C03649=1150.489,20.395,-48.948,179.944,6.210,149.138
C03650=1150.495,20.146,-48.934,179.942,6.210,149.139
C03651=1150.499,19.897,-48.920,179.939,6.209,149.139
C03652=1150.504,19.647,-48.905,179.936,6.208,149.140
C03653=1150.509,19.397,-48.891,179.934,6.207,149.141
C03654=1150.514,19.147,-48.877,179.931,6.206,149.141
C03655=1150.520,18.898,-48.863,179.929,6.205,149.142
C03656=1150.525,18.649,-48.849,179.926,6.204,149.142
C03657=1150.530,18.399,-48.834,179.924,6.203,149.143
C03658=1150.535,18.150,-48.820,179.922,6.203,149.143
C03659=1150.541,17.900,-48.807,179.919,6.202,149.144
C03660=1150.546,17.650,-48.793,179.916,6.200,149.145
C03661=1150.551,17.400,-48.778,179.914,6.200,149.145
C03662=1150.556,17.151,-48.764,179.911,6.199,149.146
C03663=1150.561,16.902,-48.750,179.909,6.199,149.146
C03664=1150.566,16.652,-48.736,179.906,6.197,149.147
C03665=1150.571,16.402,-48.722,179.903,6.197,149.147
C03666=1150.576,16.153,-48.708,179.901,6.196,149.148
C03667=1150.581,15.904,-48.694,179.898,6.195,149.149
C03668=1150.586,15.653,-48.680,179.896,6.194,149.149
C03669=1150.592,15.404,-48.667,179.894,6.193,149.150
C03670=1150.596,15.155,-48.652,179.891,6.193,149.150
C03671=1150.601,14.905,-48.638,179.889,6.192,149.151
C03672=1150.607,14.656,-48.624,179.885,6.190,149.151
C03673=1150.612,14.406,-48.611,179.883,6.190,149.152
C03674=1150.616,14.156,-48.597,179.881,6.189,149.152
C03675=1150.622,13.907,-48.583,179.878,6.188,149.153
C03676=1150.627,13.657,-48.569,179.875,6.187,149.154
C03677=1150.632,13.408,-48.554,179.873,6.186,149.154
C03678=1150.638,13.158,-48.541,179.870,6.186,149.155
C03679=1150.642,12.909,-48.527,179.868,6.185,149.155
C03680=1150.647,12.659,-48.513,179.866,6.185,149.156
C03681=1150.653,12.410,-48.499,179.863,6.183,149.156
C03682=1150.658,12.160,-48.486,179.861,6.182,149.157
C03683=1150.663,11.910,-48.471,179.858,6.182,149.158
C03684=1150.668,11.661,-48.458,179.856,6.181,149.158
C03685=1150.673,11.411,-48.445,179.853,6.180,149.159
C03686=1150.678,11.162,-48.431,179.850,6.179,149.159
C03687=1150.683,10.912,-48.416,179.848,6.178,149.160
C03688=1150.688,10.662,-48.403,179.846,6.177,149.160
C03689=1150.693,10.413,-48.390,179.843,6.177,149.161
C03690=1150.698,10.164,-48.375,179.840,6.175,149.161
C03691=1150.704,9.913,-48.362,179.838,6.175,149.162
C03692=1150.708,9.664,-48.348,179.835,6.174,149.163
C03693=1150.713,9.415,-48.334,179.833,6.174,149.163
C03694=1150.719,9.165,-48.321,179.831,6.173,149.164
C03695=1150.724,8.915,-48.307,179.827,6.172,149.164
C03696=1150.729,8.666,-48.294,179.825,6.171,149.165
C03697=1150.734,8.416,-48.280,179.823,6.170,149.165
C03698=1150.739,8.167,-48.265,179.820,6.170,149.166
C03699=1150.744,7.917,-48.253,179.818,6.169,149.166
C03700=1150.749,7.668,-48.239,179.815,6.167,149.167
C03701=1150.755,7.418,-48.225,179.813,6.167,149.168
C03702=1150.759,7.169,-48.212,179.810,6.166,149.168
C03703=1150.765,6.919,-48.198,179.808,6.165,149.169
C03704=1150.770,6.669,-48.184,179.805,6.165,149.169
C03705=1150.775,6.419,-48.171,179.802,6.163,149.170
C03706=1150.780,6.170,-48.157,179.800,6.163,149.171
C03707=1150.786,5.920,-48.144,179.798,6.162,149.171
C03708=1150.790,5.671,-48.130,179.795,6.162,149.172
C03709=1150.796,5.421,-48.117,179.793,6.161,149.172
C03710=1150.800,5.172,-48.104,179.790,6.160,149.173
C03711=1150.806,4.922,-48.090,179.787,6.159,149.173
C03712=1150.811,4.673,-48.076,179.785,6.158,149.174
C03713=1150.816,4.423,-48.063,179.783,6.158,149.175
C03714=1150.821,4.174,-48.049,179.780,6.157,149.175
C03715=1150.826,3.924,-48.036,179.778,6.156,149.176
C03716=1150.831,3.675,-48.022,179.776,6.155,149.176
C03717=1150.837,3.424,-48.009,179.772,6.154,149.177
C03718=1150.842,3.175,-47.996,179.770,6.153,149.177
C03719=1150.847,2.925,-47.982,179.767,6.153,149.178
C03720=1150.852,2.676,-47.969,179.765,6.152,149.178
C03721=1150.857,2.426,-47.955,179.763,6.152,149.179
C03722=1150.862,2.177,-47.942,179.760,6.151,149.180
C03723=1150.867,1.908,-47.927,179.757,6.150,149.180
C03724=1150.873,1.638,-47.913,179.755,6.149,149.181
C03725=1150.879,1.369,-47.899,179.752,6.148,149.181
C03726=1150.884,1.099,-47.885,179.749,6.147,149.182
C03727=1150.889,0.850,-47.871,179.747,6.146,149.183
C03728=1150.894,0.600,-47.858,179.744,6.146,149.183
C03729=1150.900,0.351,-47.845,179.742,6.145,149.184
C03730=1150.905,0.101,-47.832,179.739,6.145,149.184
C03731=1150.910,-0.148,-47.818,179.737,6.144,149.185
C03732=1150.915,-0.398,-47.805,179.734,6.143,149.186
C03733=1150.921,-0.648,-47.792,179.732,6.142,149.186
C03734=1150.925,-0.898,-47.778,179.729,6.141,149.187
C03735=1150.931,-1.147,-47.765,179.727,6.141,149.187
C03736=1150.936,-1.396,-47.752,179.724,6.140,149.188
C03737=1150.941,-1.647,-47.739,179.722,6.139,149.188
C03738=1150.946,-1.895,-47.725,179.720,6.139,149.189
C03739=1150.951,-2.146,-47.712,179.717,6.137,149.189
C03740=1150.956,-2.395,-47.699,179.715,6.136,149.190
C03741=1150.961,-2.644,-47.687,179.712,6.136,149.191
C03742=1150.967,-2.895,-47.673,179.710,6.135,149.191
C03743=1150.971,-3.143,-47.660,179.707,6.135,149.192
C03744=1150.977,-3.394,-47.646,179.705,6.134,149.192
C03745=1150.982,-3.643,-47.634,179.702,6.133,149.193
C03746=1150.988,-3.893,-47.620,179.700,6.133,149.193
C03747=1150.992,-4.143,-47.607,179.697,6.131,149.194
C03748=1150.997,-4.392,-47.595,179.695,6.131,149.195
C03749=1151.003,-4.641,-47.581,179.692,6.130,149.195
C03750=1151.007,-4.891,-47.568,179.690,6.129,149.196
C03751=1151.013,-5.140,-47.555,179.687,6.129,149.196
C03752=1151.018,-5.391,-47.542,179.685,6.128,149.197
C03753=1151.023,-5.640,-47.529,179.682,6.128,149.198
C03754=1151.029,-5.890,-47.516,179.680,6.127,149.198
C03755=1151.033,-6.140,-47.503,179.677,6.126,149.199
C03756=1151.038,-6.389,-47.490,179.675,6.125,149.199
C03757=1151.044,-6.639,-47.477,179.672,6.124,149.200
C03758=1151.049,-6.888,-47.464,179.670,6.124,149.200
C03759=1151.054,-7.137,-47.451,179.668,6.123,149.201
C03760=1151.060,-7.387,-47.438,179.665,6.122,149.202
C03761=1151.064,-7.637,-47.425,179.663,6.122,149.202
C03762=1151.069,-7.886,-47.412,179.660,6.121,149.203
C03763=1151.074,-8.136,-47.400,179.658,6.120,149.203
C03764=1151.080,-8.386,-47.386,179.655,6.120,149.204
C03765=1151.085,-8.635,-47.373,179.653,6.119,149.204
C03766=1151.090,-8.885,-47.361,179.650,6.118,149.205
C03767=1151.096,-9.134,-47.348,179.648,6.117,149.205
C03768=1151.100,-9.384,-47.335,179.645,6.117,149.206
C03769=1151.105,-9.634,-47.322,179.643,6.116,149.207
C03770=1151.110,-9.883,-47.309,179.640,6.115,149.207
C03771=1151.116,-10.133,-47.296,179.638,6.115,149.208
C03772=1151.121,-10.383,-47.283,179.635,6.114,149.208
C03773=1151.126,-10.632,-47.271,179.633,6.113,149.209
C03774=1151.131,-10.882,-47.259,179.631,6.113,149.210
C03775=1151.136,-11.132,-47.246,179.628,6.112,149.210
C03776=1151.142,-11.381,-47.233,179.626,6.111,149.211
C03777=1151.147,-11.631,-47.220,179.624,6.111,149.211
C03778=1151.152,-11.880,-47.207,179.621,6.110,149.212
C03779=1151.157,-12.130,-47.194,179.618,6.109,149.212
C03780=1151.162,-12.380,-47.181,179.616,6.108,149.213
C03781=1151.167,-12.629,-47.169,179.613,6.108,149.214
C03782=1151.173,-12.878,-47.156,179.611,6.107,149.214
C03783=1151.177,-13.128,-47.143,179.608,6.106,149.215
C03784=1151.183,-13.378,-47.131,179.606,6.105,149.215
C03785=1151.188,-13.628,-47.119,179.604,6.105,149.216
C03786=1151.194,-13.877,-47.105,179.601,6.104,149.216
C03787=1151.198,-14.127,-47.092,179.599,6.104,149.217
C03788=1151.203,-14.377,-47.080,179.597,6.103,149.218
C03789=1151.209,-14.627,-47.068,179.594,6.103,149.218
C03790=1151.214,-14.876,-47.055,179.592,6.102,149.219
C03791=1151.219,-15.125,-47.043,179.589,6.101,149.219
C03792=1151.223,-15.375,-47.030,179.587,6.101,149.220
C03793=1151.229,-15.625,-47.017,179.584,6.100,149.221
C03794=1151.235,-15.875,-47.005,179.582,6.099,149.221
C03795=1151.240,-16.124,-46.992,179.580,6.098,149.221
C03796=1151.245,-16.373,-46.980,179.577,6.097,149.222
C03797=1151.250,-16.623,-46.967,179.575,6.096,149.223
C03798=1151.255,-16.873,-46.955,179.572,6.096,149.223
C03799=1151.260,-17.123,-46.942,179.570,6.095,149.224
C03800=1151.265,-17.372,-46.929,179.567,6.095,149.225
C03801=1151.270,-17.621,-46.917,179.565,6.094,149.225
C03802=1151.276,-17.871,-46.905,179.562,6.094,149.226
C03803=1151.282,-18.121,-46.892,179.560,6.093,149.226
C03804=1151.286,-18.371,-46.879,179.557,6.092,149.227
C03805=1151.292,-18.621,-46.867,179.555,6.092,149.227
C03806=1151.297,-18.870,-46.854,179.552,6.091,149.228
C03807=1151.302,-19.119,-46.842,179.550,6.090,149.228
C03808=1151.307,-19.369,-46.830,179.548,6.090,149.229
C03809=1151.312,-19.619,-46.817,179.545,6.089,149.230
C03810=1151.317,-19.868,-46.805,179.543,6.088,149.230
C03811=1151.322,-20.119,-46.792,179.541,6.088,149.231
C03812=1151.327,-20.368,-46.780,179.538,6.087,149.231
C03813=1151.333,-20.618,-46.768,179.536,6.087,149.232
C03814=1151.338,-20.867,-46.755,179.534,6.086,149.232
C03815=1151.343,-21.117,-46.743,179.531,6.085,149.233
C03816=1151.348,-21.367,-46.731,179.529,6.085,149.234
C03817=1151.354,-21.616,-46.718,179.526,6.084,149.234
C03818=1151.359,-21.866,-46.706,179.524,6.083,149.235
C03819=1151.364,-22.115,-46.694,179.521,6.083,149.235
C03820=1151.369,-22.364,-46.681,179.519,6.082,149.236
C03821=1151.375,-22.614,-46.669,179.516,6.082,149.237
C03822=1151.379,-22.864,-46.656,179.514,6.081,149.237
C03823=1151.385,-23.114,-46.644,179.512,6.081,149.238
C03824=1151.390,-23.364,-46.632,179.509,6.080,149.238
C03825=1151.395,-23.614,-46.620,179.507,6.079,149.239
C03826=1151.400,-23.863,-46.607,179.505,6.079,149.239
C03827=1151.406,-24.133,-46.595,179.502,6.078,149.240
C03828=1151.412,-24.403,-46.582,179.499,6.076,149.241
C03829=1151.417,-24.673,-46.568,179.496,6.076,149.241
C03830=1151.423,-24.943,-46.555,179.494,6.076,149.242
C03831=1151.428,-25.192,-46.544,179.492,6.075,149.242
C03832=1151.433,-25.442,-46.531,179.489,6.074,149.243
C03833=1151.438,-25.691,-46.519,179.487,6.074,149.244
C03834=1151.443,-25.941,-46.506,179.485,6.073,149.244
C03835=1151.448,-26.191,-46.494,179.482,6.072,149.245
C03836=1151.454,-26.441,-46.482,179.480,6.072,149.245
C03837=1151.459,-26.691,-46.470,179.477,6.071,149.246
C03838=1151.464,-26.941,-46.458,179.475,6.070,149.246
C03839=1151.469,-27.190,-46.446,179.472,6.070,149.247
C03840=1151.474,-27.440,-46.434,179.470,6.069,149.248
C03841=1151.479,-27.689,-46.421,179.467,6.069,149.248
C03842=1151.485,-27.939,-46.409,179.465,6.068,149.249
C03843=1151.490,-28.189,-46.398,179.463,6.068,149.249
C03844=1151.495,-28.438,-46.385,179.460,6.067,149.250
C03845=1151.500,-28.688,-46.374,179.458,6.066,149.251
C03846=1151.505,-28.938,-46.362,179.455,6.066,149.251
C03847=1151.511,-29.187,-46.349,179.453,6.065,149.252
C03848=1151.516,-29.437,-46.337,179.451,6.064,149.252
C03849=1151.521,-29.687,-46.325,179.449,6.064,149.253
C03850=1151.526,-29.936,-46.313,179.446,6.064,149.253
C03851=1151.531,-30.186,-46.302,179.444,6.063,149.254
C03852=1151.537,-30.436,-46.290,179.442,6.063,149.255
C03853=1151.542,-30.684,-46.277,179.439,6.062,149.255
C03854=1151.548,-30.934,-46.266,179.437,6.061,149.256
C03855=1151.553,-31.184,-46.254,179.435,6.061,149.256
C03856=1151.558,-31.434,-46.242,179.432,6.060,149.257
C03857=1151.563,-31.683,-46.230,179.430,6.059,149.257
C03858=1151.569,-31.933,-46.218,179.427,6.059,149.258
C03859=1151.573,-32.183,-46.207,179.425,6.058,149.259
C03860=1151.579,-32.433,-46.195,179.423,6.057,149.259
C03861=1151.584,-32.682,-46.182,179.420,6.057,149.260
C03862=1151.589,-32.932,-46.170,179.418,6.056,149.260
C03863=1151.594,-33.181,-46.159,179.415,6.056,149.261
C03864=1151.599,-33.431,-46.147,179.413,6.055,149.261
C03865=1151.604,-33.681,-46.134,179.410,6.055,149.262
C03866=1151.609,-33.930,-46.123,179.408,6.054,149.263
C03867=1151.615,-34.180,-46.111,179.405,6.053,149.263
C03868=1151.621,-34.430,-46.100,179.403,6.053,149.264
C03869=1151.625,-34.679,-46.088,179.401,6.052,149.264
C03870=1151.631,-34.929,-46.077,179.398,6.051,149.265
C03871=1151.636,-35.178,-46.064,179.397,6.051,149.265
C03872=1151.641,-35.428,-46.052,179.394,6.051,149.266
C03873=1151.646,-35.678,-46.041,179.392,6.050,149.267
C03874=1151.651,-35.928,-46.029,179.389,6.050,149.267
C03875=1151.657,-36.178,-46.017,179.387,6.049,149.268
C03876=1151.662,-36.427,-46.006,179.384,6.049,149.268
C03877=1151.668,-36.677,-45.994,179.382,6.048,149.269
C03878=1151.672,-36.926,-45.983,179.380,6.047,149.270
C03879=1151.678,-37.176,-45.971,179.377,6.047,149.270
C03880=1151.683,-37.426,-45.958,179.375,6.046,149.271
C03881=1151.687,-37.675,-45.947,179.373,6.045,149.271
C03882=1151.693,-37.925,-45.935,179.370,6.045,149.272
C03883=1151.699,-38.174,-45.924,179.368,6.044,149.272
C03884=1151.704,-38.424,-45.912,179.366,6.044,149.273
C03885=1151.709,-38.674,-45.901,179.363,6.044,149.274
C03886=1151.714,-38.924,-45.889,179.361,6.043,149.274
C03887=1151.719,-39.174,-45.877,179.359,6.043,149.275
C03888=1151.725,-39.423,-45.866,179.356,6.042,149.275
C03889=1151.730,-39.672,-45.855,179.354,6.041,149.276
C03890=1151.735,-39.922,-45.843,179.352,6.041,149.276
C03891=1151.740,-40.172,-45.831,179.349,6.040,149.277
C03892=1151.745,-40.422,-45.820,179.347,6.039,149.278
C03893=1151.751,-40.672,-45.808,179.345,6.039,149.278
C03894=1151.756,-40.921,-45.797,179.342,6.038,149.279
C03895=1151.762,-41.171,-45.785,179.340,6.037,149.279
C03896=1151.766,-41.420,-45.774,179.338,6.038,149.280
C03897=1151.772,-41.670,-45.762,179.335,6.037,149.280
C03898=1151.776,-41.920,-45.750,179.333,6.036,149.281
C03899=1151.782,-42.169,-45.739,179.331,6.036,149.282
C03900=1151.787,-42.419,-45.728,179.328,6.035,149.282
C03901=1151.793,-42.669,-45.716,179.326,6.035,149.283
C03902=1151.798,-42.919,-45.705,179.324,6.034,149.283
C03903=1151.803,-43.169,-45.693,179.321,6.033,149.284
C03904=1151.808,-43.418,-45.682,179.319,6.033,149.284
C03905=1151.814,-43.668,-45.670,179.317,6.033,149.285
C03906=1151.818,-43.917,-45.659,179.314,6.032,149.286
C03907=1151.824,-44.167,-45.647,179.312,6.031,149.286
C03908=1151.829,-44.416,-45.636,179.310,6.031,149.287
C03909=1151.835,-44.667,-45.625,179.307,6.030,149.287
C03910=1151.840,-44.916,-45.614,179.305,6.030,149.288
C03911=1151.845,-45.166,-45.602,179.303,6.029,149.288
C03912=1151.850,-45.415,-45.591,179.300,6.029,149.289
C03913=1151.855,-45.665,-45.580,179.298,6.028,149.290
C03914=1151.860,-45.915,-45.568,179.296,6.028,149.290
C03915=1151.865,-46.165,-45.557,179.293,6.027,149.291
C03916=1151.871,-46.414,-45.546,179.291,6.027,149.291
C03917=1151.876,-46.664,-45.535,179.289,6.026,149.292
C03918=1151.882,-46.914,-45.523,179.286,6.025,149.293
C03919=1151.887,-47.163,-45.512,179.284,6.025,149.293
C03920=1151.892,-47.413,-45.501,179.282,6.024,149.294
C03921=1151.897,-47.663,-45.489,179.279,6.024,149.294
C03922=1151.902,-47.913,-45.478,179.277,6.024,149.295
C03923=1151.908,-48.162,-45.466,179.275,6.023,149.295
C03924=1151.913,-48.412,-45.456,179.272,6.023,149.296
C03925=1151.918,-48.662,-45.445,179.270,6.022,149.297
C03926=1151.924,-48.911,-45.433,179.268,6.022,149.297
C03927=1151.928,-49.161,-45.422,179.265,6.021,149.298
C03928=1151.934,-49.411,-45.411,179.263,6.020,149.298
C03929=1151.939,-49.660,-45.400,179.261,6.020,149.299
C03930=1151.944,-49.910,-45.388,179.259,6.020,149.299
C03931=1151.950,-50.181,-45.376,179.256,6.019,149.300
C03932=1151.956,-50.451,-45.364,179.254,6.019,149.301
C03933=1151.962,-50.722,-45.352,179.251,6.018,149.301
C03934=1151.967,-50.993,-45.340,179.249,6.018,149.302
C03935=1151.972,-51.242,-45.329,179.247,6.017,149.302
C03936=1151.977,-51.492,-45.318,179.244,6.016,149.303
C03937=1151.983,-51.742,-45.306,179.242,6.016,149.304
C03938=1151.988,-51.991,-45.295,179.239,6.015,149.304
C03939=1151.993,-52.241,-45.285,179.237,6.014,149.305
C03940=1151.998,-52.490,-45.274,179.235,6.014,149.305
C03941=1152.004,-52.741,-45.263,179.233,6.014,149.306
C03942=1152.009,-52.990,-45.251,179.230,6.013,149.306
C03943=1152.014,-53.239,-45.241,179.228,6.013,149.307
C03944=1152.020,-53.490,-45.229,179.226,6.012,149.308
C03945=1152.025,-53.739,-45.218,179.223,6.012,149.308
C03946=1152.030,-53.989,-45.208,179.221,6.012,149.309
C03947=1152.035,-54.239,-45.197,179.219,6.011,149.309
C03948=1152.041,-54.488,-45.186,179.216,6.010,149.310
C03949=1152.046,-54.738,-45.174,179.214,6.010,149.310
C03950=1152.051,-54.988,-45.163,179.212,6.009,149.311
C03951=1152.056,-55.237,-45.153,179.209,6.009,149.312
C03952=1152.062,-55.487,-45.141,179.208,6.009,149.312
C03953=1152.067,-55.737,-45.131,179.205,6.008,149.313
C03954=1152.072,-55.986,-45.120,179.203,6.007,149.313
C03955=1152.077,-56.237,-45.109,179.200,6.007,149.314
C03956=1152.082,-56.485,-45.098,179.198,6.006,149.315
C03957=1152.088,-56.736,-45.087,179.195,6.006,149.315
C03958=1152.093,-56.985,-45.076,179.194,6.006,149.316
C03959=1152.098,-57.235,-45.065,179.192,6.005,149.316
C03960=1152.103,-57.485,-45.054,179.189,6.005,149.317
C03961=1152.109,-57.734,-45.044,179.187,6.004,149.317
C03962=1152.113,-57.984,-45.033,179.184,6.003,149.318
C03963=1152.120,-58.234,-45.022,179.183,6.003,149.319
C03964=1152.125,-58.484,-45.011,179.180,6.003,149.319
C03965=1152.130,-58.733,-45.000,179.178,6.002,149.320
C03966=1152.135,-58.983,-44.990,179.176,6.001,149.320
C03967=1152.140,-59.232,-44.979,179.173,6.001,149.321
C03968=1152.145,-59.482,-44.968,179.171,6.001,149.321
C03969=1152.151,-59.732,-44.956,179.169,6.000,149.322
C03970=1152.156,-59.982,-44.946,179.166,6.000,149.323
C03971=1152.161,-60.232,-44.936,179.164,5.999,149.323
C03972=1152.166,-60.481,-44.925,179.162,5.999,149.324
C03973=1152.171,-60.731,-44.914,179.160,5.999,149.324
C03974=1152.177,-60.981,-44.904,179.158,5.998,149.325
C03975=1152.182,-61.230,-44.893,179.155,5.998,149.325
C03976=1152.187,-61.480,-44.882,179.153,5.997,149.326
C03977=1152.192,-61.730,-44.871,179.150,5.996,149.327
C03978=1152.198,-61.979,-44.860,179.149,5.996,149.327
C03979=1152.203,-62.230,-44.850,179.146,5.996,149.328
C03980=1152.209,-62.479,-44.839,179.144,5.995,149.328
C03981=1152.214,-62.729,-44.828,179.142,5.994,149.329
C03982=1152.219,-62.978,-44.818,179.139,5.994,149.329
C03983=1152.224,-63.229,-44.807,179.137,5.994,149.330
C03984=1152.230,-63.478,-44.797,179.135,5.993,149.330
C03985=1152.235,-63.728,-44.786,179.132,5.993,149.331
C03986=1152.240,-63.977,-44.776,179.130,5.992,149.332
C03987=1152.245,-64.227,-44.764,179.128,5.992,149.332
C03988=1152.250,-64.477,-44.754,179.126,5.992,149.333
C03989=1152.256,-64.726,-44.744,179.124,5.991,149.333
C03990=1152.261,-64.976,-44.733,179.121,5.991,149.334
C03991=1152.266,-65.225,-44.723,179.119,5.990,149.334
C03992=1152.271,-65.476,-44.712,179.117,5.990,149.335
C03993=1152.277,-65.725,-44.702,179.115,5.989,149.336
C03994=1152.282,-65.975,-44.691,179.113,5.989,149.336
C03995=1152.288,-66.225,-44.681,179.110,5.988,149.337
C03996=1152.292,-66.474,-44.670,179.108,5.988,149.337
C03997=1152.298,-66.724,-44.659,179.106,5.988,149.338
C03998=1152.303,-66.974,-44.649,179.103,5.987,149.338
C03999=1152.308,-67.224,-44.639,179.101,5.986,149.339
C04000=1152.314,-67.473,-44.628,179.099,5.986,149.340
C04001=1152.319,-67.723,-44.617,179.097,5.986,149.340
C04002=1152.324,-67.973,-44.607,179.095,5.985,149.341
C04003=1152.329,-68.223,-44.596,179.092,5.985,149.341
C04004=1152.335,-68.472,-44.586,179.090,5.984,149.342
C04005=1152.341,-68.722,-44.576,179.088,5.984,149.342
C04006=1152.346,-68.972,-44.565,179.086,5.984,149.343
C04007=1152.351,-69.222,-44.555,179.083,5.983,149.343
C04008=1152.356,-69.471,-44.544,179.081,5.982,149.344
C04009=1152.361,-69.721,-44.534,179.079,5.983,149.345
C04010=1152.367,-69.970,-44.523,179.077,5.982,149.345
C04011=1152.372,-70.221,-44.513,179.074,5.981,149.346
C04012=1152.378,-70.470,-44.503,179.072,5.981,149.346
C04013=1152.383,-70.720,-44.493,179.071,5.981,149.347
C04014=1152.388,-70.970,-44.482,179.068,5.980,149.348
C04015=1152.394,-71.219,-44.472,179.066,5.979,149.348
C04016=1152.398,-71.469,-44.462,179.063,5.979,149.349
C04017=1152.404,-71.719,-44.452,179.061,5.979,149.349
C04018=1152.409,-71.968,-44.441,179.059,5.978,149.350
C04019=1152.414,-72.219,-44.431,179.057,5.978,149.350
C04020=1152.420,-72.468,-44.421,179.054,5.977,149.351
C04021=1152.425,-72.717,-44.410,179.053,5.977,149.351
C04022=1152.430,-72.967,-44.399,179.050,5.977,149.352
C04023=1152.436,-73.217,-44.389,179.048,5.976,149.353
C04024=1152.441,-73.466,-44.379,179.045,5.976,149.353
C04025=1152.446,-73.716,-44.369,179.044,5.976,149.354
C04026=1152.451,-73.966,-44.358,179.041,5.975,149.354
C04027=1152.457,-74.216,-44.348,179.039,5.974,149.355
C04028=1152.462,-74.466,-44.338,179.037,5.974,149.355
C04029=1152.468,-74.716,-44.328,179.035,5.974,149.356
C04030=1152.473,-74.965,-44.318,179.032,5.973,149.357
C04031=1152.478,-75.215,-44.308,179.030,5.973,149.357
C04032=1152.483,-75.465,-44.298,179.029,5.973,149.358
C04033=1152.489,-75.715,-44.288,179.026,5.972,149.358
C04034=1152.494,-75.964,-44.277,179.024,5.971,149.359
C04035=1152.500,-76.235,-44.266,179.021,5.971,149.359
C04036=1152.505,-76.507,-44.255,179.019,5.970,149.360
C04037=1152.511,-76.778,-44.244,179.017,5.971,149.361
C04038=1152.517,-77.049,-44.233,179.015,5.970,149.361
C04039=1152.523,-77.299,-44.223,179.012,5.970,149.362
C04040=1152.527,-77.549,-44.213,179.010,5.969,149.362
C04041=1152.533,-77.799,-44.203,179.008,5.969,149.363
C04042=1152.539,-78.048,-44.193,179.005,5.968,149.364
C04043=1152.544,-78.299,-44.182,179.003,5.968,149.364
C04044=1152.549,-78.548,-44.172,179.001,5.967,149.364
C04045=1152.554,-78.797,-44.162,178.999,5.967,149.365
C04046=1152.560,-79.047,-44.152,178.997,5.966,149.366
C04047=1152.565,-79.298,-44.142,178.995,5.966,149.366
C04048=1152.570,-79.547,-44.132,178.992,5.966,149.367
C04049=1152.575,-79.797,-44.123,178.990,5.965,149.367
C04050=1152.581,-80.046,-44.112,178.988,5.965,149.368
C04051=1152.586,-80.296,-44.102,178.985,5.964,149.369
C04052=1152.591,-80.546,-44.092,178.984,5.964,149.369
C04053=1152.597,-80.796,-44.083,178.981,5.964,149.370
C04054=1152.602,-81.045,-44.072,178.979,5.963,149.370
C04055=1152.607,-81.296,-44.062,178.977,5.963,149.371
C04056=1152.612,-81.545,-44.052,178.975,5.963,149.371
C04057=1152.618,-81.795,-44.043,178.973,5.962,149.372
C04058=1152.624,-82.044,-44.033,178.971,5.962,149.372
C04059=1152.629,-82.294,-44.023,178.968,5.962,149.373
C04060=1152.634,-82.544,-44.012,178.966,5.961,149.374
C04061=1152.639,-82.794,-44.003,178.964,5.961,149.374
C04062=1152.644,-83.043,-43.993,178.962,5.960,149.375
C04063=1152.650,-83.293,-43.983,178.960,5.960,149.375
C04064=1152.655,-83.542,-43.973,178.957,5.959,149.376
C04065=1152.660,-83.793,-43.964,178.955,5.959,149.376
C04066=1152.666,-84.043,-43.953,178.953,5.959,149.377
C04067=1152.671,-84.292,-43.943,178.951,5.958,149.377
C04068=1152.676,-84.541,-43.934,178.949,5.958,149.378
C04069=1152.682,-84.791,-43.924,178.947,5.957,149.379
C04070=1152.686,-85.041,-43.914,178.944,5.957,149.379
C04071=1152.692,-85.291,-43.904,178.943,5.957,149.380
C04072=1152.698,-85.541,-43.894,178.940,5.956,149.380
C04073=1152.703,-85.790,-43.885,178.938,5.956,149.381
C04074=1152.708,-86.040,-43.875,178.936,5.956,149.381
C04075=1152.713,-86.290,-43.866,178.934,5.955,149.382
C04076=1152.718,-86.540,-43.855,178.932,5.954,149.382
C04077=1152.724,-86.790,-43.846,178.930,5.954,149.383
C04078=1152.729,-87.039,-43.836,178.927,5.954,149.384
C04079=1152.735,-87.289,-43.826,178.925,5.953,149.384
C04080=1152.740,-87.539,-43.817,178.924,5.953,149.385
C04081=1152.746,-87.788,-43.807,178.921,5.953,149.385
C04082=1152.750,-88.038,-43.797,178.919,5.952,149.386
C04083=1152.756,-88.288,-43.787,178.917,5.952,149.386
C04084=1152.761,-88.538,-43.777,178.914,5.952,149.387
C04085=1152.766,-88.788,-43.768,178.912,5.951,149.387
C04086=1152.772,-89.037,-43.758,178.911,5.951,149.388
C04087=1152.777,-89.287,-43.749,178.908,5.950,149.388
C04088=1152.783,-89.537,-43.739,178.906,5.950,149.389
C04089=1152.788,-89.786,-43.729,178.904,5.950,149.390
C04090=1152.793,-90.037,-43.719,178.902,5.949,149.390
C04091=1152.798,-90.286,-43.710,178.899,5.949,149.391
C04092=1152.804,-90.536,-43.700,178.898,5.949,149.391
C04093=1152.809,-90.785,-43.691,178.895,5.948,149.392
C04094=1152.814,-91.036,-43.681,178.893,5.948,149.393
C04095=1152.819,-91.285,-43.672,178.891,5.948,149.393
C04096=1152.825,-91.535,-43.662,178.889,5.947,149.393
C04097=1152.830,-91.784,-43.652,178.886,5.947,149.394
C04098=1152.836,-92.034,-43.643,178.885,5.947,149.395
C04099=1152.841,-92.284,-43.633,178.883,5.946,149.395
C04100=1152.846,-92.534,-43.623,178.881,5.946,149.396
C04101=1152.851,-92.784,-43.614,178.878,5.946,149.396
C04102=1152.857,-93.034,-43.604,178.876,5.945,149.397
C04103=1152.862,-93.283,-43.595,178.874,5.945,149.397
C04104=1152.868,-93.533,-43.585,178.872,5.944,149.398
C04105=1152.873,-93.783,-43.576,178.870,5.944,149.399
C04106=1152.878,-94.033,-43.566,178.868,5.944,149.399
C04107=1152.884,-94.283,-43.557,178.866,5.943,149.399
C04108=1152.889,-94.532,-43.548,178.863,5.943,149.400
C04109=1152.894,-94.782,-43.538,178.862,5.943,149.401
C04110=1152.899,-95.031,-43.528,178.859,5.942,149.401
C04111=1152.905,-95.281,-43.519,178.857,5.942,149.402
C04112=1152.910,-95.531,-43.510,178.855,5.941,149.402
C04113=1152.916,-95.781,-43.500,178.853,5.941,149.403
C04114=1152.921,-96.031,-43.491,178.851,5.941,149.403
C04115=1152.926,-96.280,-43.481,178.849,5.940,149.404
C04116=1152.932,-96.530,-43.472,178.846,5.940,149.405
C04117=1152.937,-96.780,-43.463,178.845,5.940,149.405
C04118=1152.943,-97.029,-43.453,178.843,5.939,149.405
C04119=1152.948,-97.279,-43.444,178.841,5.939,149.406
C04120=1152.953,-97.529,-43.435,178.838,5.939,149.407
C04121=1152.959,-97.779,-43.425,178.836,5.938,149.407
C04122=1152.964,-98.028,-43.416,178.834,5.938,149.408
C04123=1152.969,-98.278,-43.407,178.832,5.937,149.408
C04124=1152.975,-98.528,-43.397,178.830,5.937,149.409
C04125=1152.980,-98.778,-43.388,178.828,5.937,149.409
C04126=1152.986,-99.028,-43.378,178.825,5.936,149.410
C04127=1152.990,-99.277,-43.369,178.824,5.936,149.411
C04128=1152.996,-99.527,-43.360,178.822,5.936,149.411
C04129=1153.002,-99.777,-43.350,178.819,5.935,149.412
C04130=1153.007,-100.027,-43.341,178.817,5.935,149.412
C04131=1153.012,-100.276,-43.332,178.815,5.934,149.413
C04132=1153.017,-100.526,-43.322,178.814,5.934,149.413
C04133=1153.023,-100.776,-43.313,178.811,5.934,149.414
C04134=1153.028,-101.026,-43.305,178.809,5.933,149.414
C04135=1153.033,-101.276,-43.294,178.807,5.933,149.415
C04136=1153.039,-101.525,-43.285,178.805,5.933,149.415
C04137=1153.044,-101.775,-43.277,178.803,5.932,149.416
C04138=1153.049,-102.025,-43.268,178.801,5.932,149.417
C04139=1153.055,-102.297,-43.257,178.798,5.932,149.417
C04140=1153.061,-102.569,-43.247,178.796,5.931,149.418
C04141=1153.066,-102.842,-43.237,178.794,5.931,149.418
C04142=1153.072,-103.113,-43.227,178.792,5.931,149.419
C04143=1153.078,-103.363,-43.218,178.789,5.930,149.419
C04144=1153.084,-103.613,-43.209,178.788,5.930,149.420
C04145=1153.088,-103.862,-43.199,178.786,5.929,149.420
C04146=1153.094,-104.112,-43.190,178.783,5.930,149.421
C04147=1153.099,-104.362,-43.181,178.781,5.929,149.422
C04148=1153.104,-104.612,-43.173,178.779,5.928,149.422
C04149=1153.110,-104.862,-43.163,178.777,5.928,149.423
C04150=1153.115,-105.112,-43.154,178.775,5.928,149.423
C04151=1153.120,-105.361,-43.145,178.773,5.928,149.424
C04152=1153.125,-105.611,-43.136,178.771,5.927,149.424
C04153=1153.131,-105.861,-43.126,178.769,5.926,149.425
C04154=1153.137,-106.110,-43.118,178.767,5.926,149.425
C04155=1153.142,-106.360,-43.109,178.765,5.926,149.426
C04156=1153.147,-106.610,-43.100,178.763,5.926,149.426
C04157=1153.152,-106.860,-43.091,178.761,5.925,149.427
C04158=1153.158,-107.110,-43.081,178.759,5.925,149.427
C04159=1153.163,-107.360,-43.073,178.756,5.925,149.428
C04160=1153.168,-107.609,-43.063,178.754,5.924,149.429
C04161=1153.173,-107.859,-43.054,178.753,5.924,149.429
C04162=1153.178,-108.109,-43.045,178.750,5.924,149.430
C04163=1153.185,-108.358,-43.036,178.749,5.924,149.430
C04164=1153.190,-108.608,-43.027,178.746,5.923,149.431
C04165=1153.195,-108.858,-43.018,178.744,5.922,149.431
C04166=1153.200,-109.108,-43.009,178.742,5.923,149.432
C04167=1153.206,-109.358,-43.000,178.740,5.922,149.432
C04168=1153.211,-109.608,-42.992,178.738,5.922,149.433
C04169=1153.217,-109.858,-42.982,178.736,5.921,149.433
C04170=1153.222,-110.108,-42.973,178.734,5.921,149.434
C04171=1153.228,-110.357,-42.965,178.732,5.921,149.434
C04172=1153.233,-110.607,-42.956,178.731,5.921,149.435
C04173=1153.238,-110.856,-42.947,178.728,5.920,149.436
C04174=1153.243,-111.106,-42.938,178.726,5.920,149.436
C04175=1153.248,-111.356,-42.929,178.724,5.920,149.437
C04176=1153.253,-111.606,-42.920,178.722,5.919,149.437
C04177=1153.260,-111.855,-42.911,178.720,5.919,149.438
C04178=1153.265,-112.105,-42.902,178.718,5.919,149.438
C04179=1153.270,-112.355,-42.893,178.716,5.919,149.439
C04180=1153.275,-112.605,-42.884,178.714,5.918,149.439
C04181=1153.281,-112.855,-42.875,178.712,5.917,149.440
C04182=1153.286,-113.104,-42.867,178.710,5.917,149.440
C04183=1153.292,-113.354,-42.858,178.707,5.917,149.441
C04184=1153.297,-113.604,-42.849,178.706,5.917,149.441
C04185=1153.302,-113.854,-42.841,178.704,5.916,149.442
C04186=1153.307,-114.104,-42.832,178.702,5.916,149.442
C04187=1153.313,-114.353,-42.823,178.700,5.915,149.443
C04188=1153.318,-114.603,-42.815,178.698,5.916,149.444
C04189=1153.324,-114.853,-42.805,178.695,5.915,149.444
C04190=1153.329,-115.103,-42.796,178.694,5.915,149.445
C04191=1153.335,-115.353,-42.787,178.692,5.914,149.445
C04192=1153.340,-115.602,-42.779,178.689,5.914,149.446
C04193=1153.345,-115.852,-42.770,178.687,5.914,149.446
C04194=1153.351,-116.102,-42.762,178.685,5.913,149.447
C04195=1153.356,-116.352,-42.753,178.684,5.913,149.447
C04196=1153.362,-116.601,-42.744,178.681,5.912,149.448
C04197=1153.367,-116.851,-42.735,178.680,5.913,149.448
C04198=1153.372,-117.101,-42.726,178.678,5.912,149.449
C04199=1153.377,-117.351,-42.718,178.676,5.912,149.449
C04200=1153.383,-117.601,-42.709,178.673,5.911,149.450
C04201=1153.389,-117.850,-42.701,178.672,5.911,149.450
C04202=1153.394,-118.100,-42.692,178.670,5.911,149.451
C04203=1153.399,-118.350,-42.683,178.667,5.910,149.451
C04204=1153.404,-118.600,-42.674,178.666,5.910,149.452
C04205=1153.410,-118.850,-42.666,178.663,5.910,149.453
C04206=1153.415,-119.100,-42.657,178.662,5.910,149.453
C04207=1153.421,-119.349,-42.649,178.659,5.909,149.454
C04208=1153.426,-119.599,-42.640,178.658,5.909,149.454
C04209=1153.431,-119.848,-42.631,178.656,5.908,149.455
C04210=1153.437,-120.099,-42.623,178.654,5.908,149.455
C04211=1153.442,-120.349,-42.614,178.651,5.908,149.456
C04212=1153.448,-120.598,-42.605,178.650,5.908,149.456
C04213=1153.452,-120.848,-42.597,178.647,5.907,149.457
C04214=1153.458,-121.098,-42.589,178.646,5.907,149.457
C04215=1153.463,-121.348,-42.580,178.644,5.906,149.458
C04216=1153.469,-121.597,-42.572,178.642,5.907,149.458
C04217=1153.474,-121.847,-42.563,178.639,5.906,149.459
C04218=1153.479,-122.097,-42.554,178.638,5.906,149.459
C04219=1153.485,-122.346,-42.546,178.636,5.905,149.460
C04220=1153.490,-122.596,-42.537,178.634,5.905,149.460
C04221=1153.496,-122.847,-42.529,178.632,5.905,149.461
C04222=1153.502,-123.096,-42.520,178.630,5.905,149.461
C04223=1153.507,-123.346,-42.511,178.628,5.904,149.462
C04224=1153.512,-123.596,-42.503,178.626,5.904,149.462
C04225=1153.517,-123.845,-42.495,178.624,5.904,149.463
C04226=1153.522,-124.095,-42.486,178.622,5.904,149.463
C04227=1153.528,-124.345,-42.478,178.620,5.903,149.464
C04228=1153.534,-124.595,-42.470,178.618,5.902,149.464
C04229=1153.539,-124.844,-42.461,178.616,5.902,149.465
C04230=1153.544,-125.095,-42.453,178.614,5.902,149.465
C04231=1153.550,-125.344,-42.444,178.612,5.902,149.466
C04232=1153.555,-125.594,-42.435,178.610,5.901,149.467
C04233=1153.560,-125.844,-42.428,178.608,5.901,149.467
C04234=1153.566,-126.093,-42.419,178.606,5.900,149.468
C04235=1153.571,-126.344,-42.411,178.604,5.901,149.468
C04236=1153.576,-126.594,-42.402,178.602,5.900,149.469
C04237=1153.582,-126.843,-42.393,178.600,5.900,149.469
C04238=1153.588,-127.093,-42.385,178.598,5.899,149.470
C04239=1153.592,-127.343,-42.377,178.596,5.900,149.470
C04240=1153.598,-127.592,-42.369,178.594,5.899,149.471
C04241=1153.603,-127.842,-42.360,178.592,5.899,149.471
C04242=1153.609,-128.093,-42.352,178.590,5.898,149.472
C04243=1153.188,-128.103,-42.394,178.587,5.902,149.474
C04244=1153.182,-127.854,-42.403,178.589,5.902,149.473
C04245=1153.177,-127.604,-42.412,178.591,5.902,149.472
C04246=1153.171,-127.353,-42.420,178.593,5.902,149.472
C04247=1153.166,-127.105,-42.428,178.595,5.903,149.471
C04248=1153.161,-126.854,-42.436,178.597,5.903,149.471
C04249=1153.156,-126.604,-42.445,178.599,5.904,149.470
C04250=1153.150,-126.355,-42.453,178.600,5.904,149.470
C04251=1153.144,-126.105,-42.462,178.603,5.905,149.469
C04252=1153.139,-125.855,-42.470,178.604,5.905,149.469
C04253=1153.134,-125.605,-42.478,178.606,5.905,149.468
C04254=1153.129,-125.356,-42.487,178.608,5.905,149.468
C04255=1153.123,-125.105,-42.495,178.611,5.906,149.467
C04256=1153.118,-124.856,-42.503,178.612,5.906,149.467
C04257=1153.112,-124.606,-42.512,178.614,5.906,149.466
C04258=1153.107,-124.356,-42.520,178.616,5.906,149.466
C04259=1153.101,-124.106,-42.529,178.618,5.907,149.465
C04260=1153.097,-123.857,-42.537,178.620,5.907,149.465
C04261=1153.091,-123.606,-42.545,178.623,5.907,149.464
C04262=1153.085,-123.357,-42.554,178.624,5.907,149.464
C04263=1153.080,-123.107,-42.563,178.626,5.908,149.463
C04264=1153.075,-122.857,-42.571,178.628,5.908,149.463
C04265=1153.069,-122.608,-42.579,178.630,5.909,149.462
C04266=1153.064,-122.358,-42.588,178.632,5.909,149.462
C04267=1153.058,-122.107,-42.597,178.634,5.909,149.461
C04268=1153.053,-121.858,-42.605,178.637,5.910,149.460
C04269=1153.047,-121.608,-42.614,178.638,5.910,149.460
C04270=1153.042,-121.359,-42.623,178.640,5.911,149.459
C04271=1153.038,-121.108,-42.630,178.642,5.910,149.459
C04272=1153.032,-120.859,-42.639,178.644,5.911,149.458
C04273=1153.027,-120.609,-42.648,178.646,5.911,149.458
C04274=1153.021,-120.360,-42.657,178.648,5.912,149.458
C04275=1153.015,-120.110,-42.665,178.650,5.912,149.457
C04276=1153.010,-119.860,-42.674,178.652,5.912,149.456
C04277=1153.005,-119.610,-42.682,178.654,5.912,149.456
C04278=1153.000,-119.360,-42.691,178.656,5.913,149.455
C04279=1152.994,-119.111,-42.699,178.658,5.913,149.455
C04280=1152.989,-118.861,-42.708,178.660,5.914,149.454
C04281=1152.983,-118.611,-42.717,178.662,5.913,149.454
C04282=1152.978,-118.361,-42.726,178.664,5.914,149.453
C04283=1152.973,-118.112,-42.734,178.666,5.914,149.453
C04284=1152.967,-117.861,-42.743,178.668,5.915,149.452
C04285=1152.962,-117.612,-42.751,178.670,5.915,149.452
C04286=1152.957,-117.362,-42.760,178.672,5.915,149.451
C04287=1152.951,-117.113,-42.769,178.674,5.916,149.451
C04288=1152.946,-116.863,-42.778,178.676,5.916,149.450
C04289=1152.940,-116.612,-42.786,178.678,5.917,149.450
C04290=1152.935,-116.362,-42.795,178.680,5.916,149.449
C04291=1152.929,-116.113,-42.803,178.682,5.917,149.449
C04292=1152.924,-115.863,-42.812,178.684,5.917,149.448
C04293=1152.919,-115.613,-42.821,178.686,5.918,149.447
C04294=1152.914,-115.364,-42.830,178.688,5.918,149.447
C04295=1152.908,-115.114,-42.839,178.690,5.918,149.446
C04296=1152.903,-114.865,-42.848,178.692,5.918,149.446
C04297=1152.897,-114.614,-42.856,178.694,5.919,149.445
C04298=1152.892,-114.364,-42.865,178.697,5.919,149.445
C04299=1152.887,-114.114,-42.873,178.698,5.919,149.444
C04300=1152.881,-113.865,-42.883,178.700,5.920,149.444
C04301=1152.875,-113.615,-42.892,178.702,5.920,149.443
C04302=1152.870,-113.365,-42.900,178.704,5.921,149.443
C04303=1152.865,-113.115,-42.909,178.706,5.920,149.442
C04304=1152.860,-112.866,-42.918,178.708,5.921,149.442
C04305=1152.854,-112.616,-42.927,178.710,5.921,149.441
C04306=1152.849,-112.367,-42.936,178.712,5.922,149.441
C04307=1152.844,-112.117,-42.945,178.714,5.923,149.440
C04308=1152.839,-111.867,-42.953,178.716,5.923,149.440
C04309=1152.834,-111.617,-42.962,178.719,5.923,149.439
C04310=1152.828,-111.368,-42.971,178.720,5.923,149.438
C04311=1152.822,-111.118,-42.980,178.722,5.924,149.438
C04312=1152.816,-110.867,-42.989,178.724,5.924,149.437
C04313=1152.811,-110.617,-42.997,178.726,5.924,149.437
C04314=1152.806,-110.368,-43.006,178.728,5.924,149.436
C04315=1152.801,-110.118,-43.015,178.730,5.925,149.436
C04316=1152.796,-109.868,-43.024,178.733,5.925,149.435
C04317=1152.790,-109.619,-43.033,178.734,5.925,149.435
C04318=1152.784,-109.369,-43.043,178.737,5.926,149.434
C04319=1152.779,-109.119,-43.052,178.739,5.926,149.434
C04320=1152.774,-108.869,-43.061,178.741,5.927,149.433
C04321=1152.769,-108.620,-43.070,178.742,5.926,149.433
C04322=1152.764,-108.370,-43.078,178.745,5.927,149.432
C04323=1152.759,-108.120,-43.087,178.747,5.928,149.431
C04324=1152.752,-107.870,-43.096,178.749,5.928,149.431
C04325=1152.747,-107.621,-43.105,178.751,5.928,149.430
C04326=1152.742,-107.371,-43.114,178.753,5.928,149.430
C04327=1152.737,-107.121,-43.123,178.755,5.929,149.429
C04328=1152.731,-106.871,-43.132,178.757,5.929,149.429
C04329=1152.726,-106.621,-43.141,178.759,5.929,149.428
C04330=1152.720,-106.371,-43.150,178.761,5.930,149.428
C04331=1152.715,-106.121,-43.159,178.763,5.930,149.427
C04332=1152.710,-105.872,-43.169,178.766,5.930,149.427
C04333=1152.705,-105.623,-43.178,178.767,5.930,149.426
C04334=1152.699,-105.373,-43.186,178.769,5.931,149.426
C04335=1152.693,-105.123,-43.196,178.772,5.932,149.425
C04336=1152.688,-104.873,-43.205,178.774,5.932,149.424
C04337=1152.683,-104.623,-43.214,178.776,5.932,149.424
C04338=1152.678,-104.373,-43.223,178.777,5.932,149.423
C04339=1152.672,-104.124,-43.233,178.780,5.933,149.423
C04340=1152.667,-103.874,-43.242,178.782,5.933,149.422
C04341=1152.662,-103.624,-43.251,178.784,5.933,149.422
C04342=1152.657,-103.374,-43.260,178.786,5.934,149.421
C04343=1152.651,-103.124,-43.269,178.788,5.934,149.421
C04344=1152.645,-102.852,-43.279,178.790,5.934,149.420
C04345=1152.639,-102.581,-43.289,178.793,5.935,149.420
C04346=1152.634,-102.308,-43.299,178.795,5.936,149.419
C04347=1152.628,-102.036,-43.309,178.797,5.936,149.418
C04348=1152.622,-101.786,-43.318,178.799,5.936,149.418
C04349=1152.617,-101.536,-43.327,178.802,5.937,149.417
C04350=1152.612,-101.287,-43.337,178.803,5.937,149.417
C04351=1152.607,-101.037,-43.346,178.805,5.937,149.416
C04352=1152.601,-100.787,-43.355,178.807,5.937,149.416
C04353=1152.596,-100.537,-43.364,178.810,5.938,149.415
C04354=1152.591,-100.288,-43.374,178.812,5.938,149.415
C04355=1152.585,-100.038,-43.383,178.814,5.938,149.414
C04356=1152.580,-99.788,-43.392,178.816,5.939,149.414
C04357=1152.575,-99.538,-43.401,178.818,5.939,149.413
C04358=1152.569,-99.289,-43.411,178.820,5.940,149.412
C04359=1152.564,-99.039,-43.420,178.822,5.940,149.412
C04360=1152.559,-98.789,-43.429,178.824,5.940,149.411
C04361=1152.553,-98.539,-43.439,178.826,5.941,149.411
C04362=1152.548,-98.289,-43.448,178.828,5.941,149.410
C04363=1152.543,-98.040,-43.457,178.830,5.941,149.410
C04364=1152.537,-97.790,-43.467,178.832,5.942,149.409
C04365=1152.532,-97.540,-43.476,178.835,5.942,149.409
C04366=1152.526,-97.290,-43.486,178.837,5.943,149.408
C04367=1152.521,-97.041,-43.495,178.839,5.943,149.408
C04368=1152.516,-96.791,-43.504,178.840,5.943,149.407
C04369=1152.510,-96.541,-43.514,178.843,5.944,149.406
C04370=1152.505,-96.292,-43.523,178.845,5.944,149.406
C04371=1152.500,-96.041,-43.533,178.847,5.944,149.405
C04372=1152.494,-95.792,-43.542,178.850,5.945,149.405
C04373=1152.490,-95.542,-43.551,178.851,5.945,149.404
C04374=1152.484,-95.292,-43.561,178.853,5.945,149.404
C04375=1152.479,-95.043,-43.570,178.856,5.946,149.403
C04376=1152.473,-94.793,-43.580,178.858,5.946,149.402
C04377=1152.468,-94.543,-43.589,178.860,5.947,149.402
C04378=1152.462,-94.293,-43.599,178.862,5.947,149.402
C04379=1152.457,-94.044,-43.608,178.864,5.947,149.401
C04380=1152.452,-93.794,-43.617,178.866,5.948,149.400
C04381=1152.446,-93.544,-43.627,178.868,5.948,149.400
C04382=1152.441,-93.295,-43.637,178.870,5.948,149.399
C04383=1152.435,-93.045,-43.646,178.873,5.949,149.399
C04384=1152.430,-92.795,-43.655,178.874,5.949,149.398
C04385=1152.425,-92.545,-43.666,178.877,5.950,149.398
C04386=1152.420,-92.295,-43.674,178.879,5.950,149.397
C04387=1152.414,-92.045,-43.685,178.881,5.950,149.396
C04388=1152.409,-91.795,-43.694,178.883,5.951,149.396
C04389=1152.404,-91.546,-43.704,178.885,5.951,149.396
C04390=1152.399,-91.296,-43.713,178.887,5.951,149.395
C04391=1152.393,-91.046,-43.723,178.890,5.952,149.394
C04392=1152.388,-90.797,-43.732,178.892,5.953,149.394
C04393=1152.382,-90.547,-43.742,178.894,5.952,149.393
C04394=1152.377,-90.297,-43.751,178.896,5.953,149.393
C04395=1152.371,-90.048,-43.761,178.898,5.954,149.392
C04396=1152.367,-89.798,-43.771,178.900,5.954,149.392
C04397=1152.361,-89.548,-43.781,178.902,5.954,149.391
C04398=1152.356,-89.298,-43.790,178.905,5.955,149.390
C04399=1152.350,-89.048,-43.800,178.906,5.955,149.390
C04400=1152.346,-88.799,-43.809,178.909,5.955,149.389
C04401=1152.340,-88.549,-43.819,178.911,5.955,149.389
C04402=1152.335,-88.300,-43.828,178.913,5.956,149.388
C04403=1152.329,-88.049,-43.838,178.915,5.956,149.388
C04404=1152.324,-87.799,-43.848,178.917,5.956,149.387
C04405=1152.319,-87.550,-43.858,178.919,5.957,149.387
C04406=1152.313,-87.300,-43.868,178.921,5.958,149.386
C04407=1152.308,-87.051,-43.877,178.923,5.957,149.385
C04408=1152.303,-86.801,-43.887,178.926,5.958,149.385
C04409=1152.298,-86.551,-43.896,178.928,5.959,149.384
C04410=1152.293,-86.301,-43.907,178.931,5.959,149.384
C04411=1152.287,-86.051,-43.916,178.932,5.959,149.383
C04412=1152.282,-85.802,-43.926,178.934,5.960,149.383
C04413=1152.276,-85.552,-43.936,178.937,5.960,149.382
C04414=1152.271,-85.302,-43.945,178.939,5.960,149.382
C04415=1152.265,-85.053,-43.955,178.941,5.961,149.381
C04416=1152.260,-84.802,-43.966,178.943,5.961,149.380
C04417=1152.255,-84.552,-43.975,178.945,5.961,149.380
C04418=1152.250,-84.303,-43.985,178.947,5.962,149.379
C04419=1152.244,-84.053,-43.995,178.950,5.963,149.379
C04420=1152.239,-83.804,-44.005,178.951,5.963,149.378
C04421=1152.234,-83.553,-44.015,178.954,5.963,149.378
C04422=1152.229,-83.304,-44.024,178.956,5.964,149.377
C04423=1152.223,-83.055,-44.034,178.958,5.964,149.377
C04424=1152.218,-82.804,-44.044,178.960,5.964,149.376
C04425=1152.213,-82.555,-44.054,178.963,5.965,149.375
C04426=1152.208,-82.305,-44.064,178.964,5.965,149.375
C04427=1152.202,-82.055,-44.074,178.967,5.966,149.374
C04428=1152.196,-81.805,-44.084,178.969,5.966,149.374
C04429=1152.191,-81.556,-44.093,178.971,5.967,149.373
C04430=1152.186,-81.306,-44.104,178.973,5.967,149.373
C04431=1152.181,-81.056,-44.114,178.976,5.967,149.372
C04432=1152.176,-80.807,-44.124,178.978,5.968,149.372
C04433=1152.170,-80.557,-44.133,178.979,5.968,149.371
C04434=1152.164,-80.307,-44.144,178.982,5.968,149.370
C04435=1152.160,-80.057,-44.154,178.984,5.969,149.370
C04436=1152.155,-79.808,-44.164,178.986,5.969,149.369
C04437=1152.149,-79.558,-44.174,178.989,5.969,149.369
C04438=1152.143,-79.308,-44.183,178.991,5.970,149.368
C04439=1152.139,-79.058,-44.193,178.993,5.971,149.368
C04440=1152.133,-78.809,-44.204,178.995,5.970,149.367
C04441=1152.128,-78.559,-44.214,178.997,5.971,149.367
C04442=1152.122,-78.309,-44.224,178.999,5.972,149.366
C04443=1152.118,-78.060,-44.234,179.002,5.972,149.365
C04444=1152.112,-77.810,-44.244,179.004,5.972,149.365
C04445=1152.106,-77.560,-44.254,179.006,5.973,149.364
C04446=1152.101,-77.310,-44.264,179.009,5.974,149.364
C04447=1152.096,-77.060,-44.275,179.010,5.973,149.363
C04448=1152.090,-76.789,-44.285,179.013,5.974,149.362
C04449=1152.085,-76.518,-44.296,179.015,5.975,149.362
C04450=1152.079,-76.247,-44.308,179.018,5.975,149.361
C04451=1152.073,-75.976,-44.318,179.020,5.976,149.361
C04452=1152.068,-75.726,-44.329,179.022,5.975,149.360
C04453=1152.062,-75.476,-44.339,179.024,5.976,149.360
C04454=1152.056,-75.226,-44.348,179.026,5.977,149.359
C04455=1152.051,-74.976,-44.359,179.029,5.977,149.358
C04456=1152.046,-74.726,-44.369,179.031,5.977,149.358
C04457=1152.041,-74.477,-44.379,179.033,5.978,149.357
C04458=1152.036,-74.227,-44.389,179.036,5.978,149.357
C04459=1152.030,-73.977,-44.400,179.038,5.979,149.356
C04460=1152.025,-73.728,-44.410,179.039,5.979,149.356
C04461=1152.020,-73.477,-44.420,179.042,5.980,149.355
C04462=1152.014,-73.228,-44.431,179.044,5.980,149.355
C04463=1152.009,-72.978,-44.441,179.046,5.980,149.354
C04464=1152.004,-72.728,-44.451,179.048,5.981,149.353
C04465=1151.999,-72.479,-44.461,179.051,5.982,149.353
C04466=1151.993,-72.229,-44.471,179.053,5.982,149.352
C04467=1151.988,-71.979,-44.482,179.055,5.982,149.352
C04468=1151.983,-71.730,-44.492,179.057,5.983,149.351
C04469=1151.977,-71.480,-44.502,179.060,5.983,149.351
C04470=1151.972,-71.230,-44.513,179.062,5.984,149.350
C04471=1151.967,-70.981,-44.524,179.064,5.984,149.350
C04472=1151.961,-70.731,-44.534,179.066,5.984,149.349
C04473=1151.956,-70.481,-44.544,179.068,5.985,149.348
C04474=1151.951,-70.232,-44.554,179.071,5.986,149.348
C04475=1151.946,-69.982,-44.565,179.073,5.985,149.347
C04476=1151.941,-69.732,-44.575,179.075,5.986,149.347
C04477=1151.935,-69.482,-44.585,179.078,5.986,149.346
C04478=1151.930,-69.232,-44.596,179.080,5.987,149.346
C04479=1151.924,-68.983,-44.606,179.081,5.987,149.345
C04480=1151.919,-68.733,-44.616,179.084,5.988,149.344
C04481=1151.914,-68.483,-44.627,179.086,5.988,149.344
C04482=1151.908,-68.234,-44.638,179.088,5.989,149.343
C04483=1151.903,-67.984,-44.648,179.090,5.989,149.343
C04484=1151.898,-67.734,-44.658,179.093,5.990,149.342
C04485=1151.893,-67.484,-44.669,179.095,5.990,149.341
C04486=1151.887,-67.234,-44.679,179.097,5.991,149.341
C04487=1151.882,-66.985,-44.690,179.100,5.991,149.341
C04488=1151.877,-66.735,-44.701,179.102,5.991,149.340
C04489=1151.871,-66.486,-44.711,179.104,5.992,149.339
C04490=1151.866,-66.235,-44.721,179.106,5.993,149.339
C04491=1151.861,-65.986,-44.732,179.109,5.993,149.338
C04492=1151.856,-65.736,-44.743,179.110,5.993,149.338
C04493=1151.851,-65.487,-44.753,179.113,5.993,149.337
C04494=1151.845,-65.237,-44.763,179.115,5.994,149.336
C04495=1151.840,-64.987,-44.774,179.117,5.995,149.336
C04496=1151.835,-64.738,-44.785,179.120,5.995,149.335
C04497=1151.830,-64.488,-44.795,179.122,5.995,149.335
C04498=1151.824,-64.238,-44.806,179.124,5.996,149.334
C04499=1151.819,-63.988,-44.816,179.127,5.997,149.334
C04500=1151.814,-63.739,-44.827,179.129,5.997,149.333
C04501=1151.809,-63.489,-44.838,179.131,5.997,149.332
C04502=1151.803,-63.239,-44.848,179.133,5.998,149.332
C04503=1151.798,-62.989,-44.858,179.136,5.998,149.331
C04504=1151.793,-62.740,-44.869,179.138,5.999,149.331
C04505=1151.788,-62.490,-44.880,179.140,6.000,149.330
C04506=1151.782,-62.240,-44.891,179.142,5.999,149.330
C04507=1151.777,-61.990,-44.902,179.144,6.000,149.329
C04508=1151.771,-61.741,-44.912,179.146,6.001,149.329
C04509=1151.766,-61.491,-44.923,179.149,6.001,149.328
C04510=1151.761,-61.242,-44.934,179.151,6.002,149.327
C04511=1151.756,-60.991,-44.944,179.153,6.002,149.327
C04512=1151.750,-60.742,-44.955,179.156,6.002,149.326
C04513=1151.746,-60.492,-44.966,179.158,6.003,149.326
C04514=1151.740,-60.243,-44.976,179.160,6.003,149.325
C04515=1151.735,-59.993,-44.987,179.163,6.004,149.325
C04516=1151.729,-59.743,-44.998,179.165,6.004,149.324
C04517=1151.724,-59.493,-45.009,179.167,6.005,149.323
C04518=1151.719,-59.244,-45.020,179.169,6.005,149.323
C04519=1151.714,-58.994,-45.030,179.172,6.006,149.322
C04520=1151.708,-58.745,-45.041,179.174,6.007,149.322
C04521=1151.703,-58.495,-45.052,179.176,6.006,149.321
C04522=1151.698,-58.244,-45.062,179.178,6.007,149.321
C04523=1151.692,-57.995,-45.074,179.180,6.008,149.320
C04524=1151.687,-57.745,-45.084,179.183,6.008,149.319
C04525=1151.682,-57.496,-45.095,179.185,6.009,149.319
C04526=1151.677,-57.246,-45.106,179.187,6.009,149.318
C04527=1151.672,-56.997,-45.117,179.190,6.009,149.318
C04528=1151.666,-56.746,-45.128,179.192,6.010,149.317
C04529=1151.661,-56.497,-45.139,179.194,6.011,149.317
C04530=1151.656,-56.247,-45.149,179.197,6.011,149.316
C04531=1151.651,-55.997,-45.161,179.199,6.012,149.315
C04532=1151.646,-55.748,-45.171,179.201,6.012,149.315
C04533=1151.640,-55.498,-45.183,179.204,6.012,149.314
C04534=1151.635,-55.248,-45.193,179.206,6.013,149.314
C04535=1151.630,-54.999,-45.204,179.208,6.014,149.313
C04536=1151.625,-54.749,-45.215,179.211,6.014,149.313
C04537=1151.620,-54.500,-45.226,179.213,6.015,149.312
C04538=1151.614,-54.250,-45.238,179.215,6.014,149.311
C04539=1151.609,-53.999,-45.248,179.217,6.015,149.311
C04540=1151.604,-53.751,-45.259,179.219,6.016,149.310
C04541=1151.599,-53.500,-45.270,179.222,6.016,149.310
C04542=1151.593,-53.251,-45.281,179.224,6.017,149.309
C04543=1151.588,-53.001,-45.292,179.227,6.018,149.308
C04544=1151.583,-52.751,-45.303,179.228,6.018,149.308
C04545=1151.577,-52.502,-45.315,179.231,6.018,149.307
C04546=1151.572,-52.252,-45.325,179.233,6.019,149.307
C04547=1151.567,-52.002,-45.337,179.235,6.020,149.306
C04548=1151.561,-51.752,-45.347,179.238,6.020,149.306
C04549=1151.556,-51.503,-45.359,179.240,6.021,149.305
C04550=1151.551,-51.254,-45.370,179.243,6.021,149.304
C04551=1151.546,-51.003,-45.380,179.244,6.021,149.304
C04552=1151.540,-50.732,-45.392,179.247,6.022,149.303
C04553=1151.535,-50.463,-45.405,179.249,6.022,149.303
C04554=1151.529,-50.192,-45.417,179.252,6.023,149.302
C04555=1151.523,-49.921,-45.430,179.255,6.023,149.301
C04556=1151.518,-49.671,-45.440,179.257,6.024,149.301
C04557=1151.513,-49.422,-45.451,179.259,6.025,149.300
C04558=1151.508,-49.172,-45.463,179.262,6.025,149.300
C04559=1151.502,-48.923,-45.474,179.264,6.026,149.299
C04560=1151.497,-48.672,-45.485,179.267,6.026,149.299
C04561=1151.492,-48.423,-45.496,179.269,6.027,149.298
C04562=1151.487,-48.174,-45.507,179.270,6.027,149.298
C04563=1151.481,-47.923,-45.518,179.273,6.027,149.297
C04564=1151.476,-47.674,-45.530,179.275,6.028,149.296
C04565=1151.470,-47.424,-45.541,179.278,6.029,149.296
C04566=1151.465,-47.175,-45.552,179.280,6.029,149.295
C04567=1151.460,-46.924,-45.563,179.283,6.030,149.295
C04568=1151.455,-46.674,-45.575,179.285,6.031,149.294
C04569=1151.450,-46.426,-45.586,179.287,6.031,149.294
C04570=1151.444,-46.176,-45.598,179.289,6.031,149.293
C04571=1151.440,-45.926,-45.609,179.291,6.032,149.292
C04572=1151.433,-45.676,-45.620,179.294,6.032,149.292
C04573=1151.429,-45.427,-45.631,179.296,6.033,149.291
C04574=1151.424,-45.177,-45.642,179.299,6.033,149.291
C04575=1151.418,-44.927,-45.654,179.301,6.034,149.290
C04576=1151.413,-44.678,-45.665,179.304,6.035,149.289
C04577=1151.408,-44.428,-45.677,179.306,6.035,149.289
C04578=1151.403,-44.178,-45.688,179.307,6.035,149.288
C04579=1151.397,-43.928,-45.700,179.310,6.036,149.288
C04580=1151.392,-43.679,-45.710,179.312,6.037,149.287
C04581=1151.387,-43.429,-45.722,179.315,6.037,149.287
C04582=1151.382,-43.179,-45.734,179.317,6.038,149.286
C04583=1151.376,-42.929,-45.746,179.320,6.038,149.285
C04584=1151.372,-42.680,-45.757,179.322,6.039,149.285
C04585=1151.366,-42.431,-45.768,179.324,6.040,149.284
C04586=1151.361,-42.181,-45.780,179.327,6.040,149.284
C04587=1151.356,-41.931,-45.792,179.329,6.041,149.283
C04588=1151.351,-41.681,-45.803,179.331,6.041,149.283
C04589=1151.345,-41.432,-45.814,179.333,6.041,149.282
C04590=1151.340,-41.182,-45.825,179.336,6.042,149.281
C04591=1151.334,-40.932,-45.837,179.338,6.043,149.281
C04592=1151.330,-40.682,-45.848,179.340,6.043,149.280
C04593=1151.324,-40.432,-45.860,179.343,6.044,149.280
C04594=1151.318,-40.183,-45.872,179.345,6.045,149.279
C04595=1151.314,-39.934,-45.883,179.348,6.045,149.279
C04596=1151.308,-39.684,-45.895,179.350,6.046,149.278
C04597=1151.303,-39.434,-45.906,179.353,6.046,149.277
C04598=1151.298,-39.184,-45.918,179.355,6.047,149.277
C04599=1151.293,-38.934,-45.929,179.357,6.047,149.276
C04600=1151.287,-38.685,-45.941,179.359,6.047,149.276
C04601=1151.282,-38.435,-45.953,179.361,6.048,149.275
C04602=1151.277,-38.186,-45.964,179.364,6.049,149.275
C04603=1151.272,-37.936,-45.976,179.366,6.049,149.274
C04604=1151.267,-37.687,-45.988,179.369,6.050,149.273
C04605=1151.262,-37.437,-46.000,179.371,6.051,149.273
C04606=1151.256,-37.188,-46.011,179.374,6.051,149.272
C04607=1151.251,-36.938,-46.022,179.376,6.052,149.272
C04608=1151.246,-36.688,-46.034,179.379,6.052,149.271
C04609=1151.240,-36.438,-46.046,179.381,6.053,149.271
C04610=1151.236,-36.188,-46.057,179.383,6.054,149.270
C04611=1151.230,-35.938,-46.069,179.386,6.054,149.269
C04612=1151.225,-35.689,-46.081,179.387,6.054,149.269
C04613=1151.220,-35.439,-46.093,179.390,6.055,149.268
C04614=1151.214,-35.190,-46.105,179.392,6.055,149.268
C04615=1151.209,-34.940,-46.117,179.395,6.056,149.267
C04616=1151.204,-34.691,-46.128,179.397,6.057,149.267
C04617=1151.199,-34.441,-46.140,179.400,6.057,149.266
C04618=1151.193,-34.191,-46.152,179.402,6.058,149.265
C04619=1151.189,-33.941,-46.163,179.404,6.058,149.265
C04620=1151.183,-33.691,-46.175,179.407,6.059,149.264
C04621=1151.178,-33.442,-46.187,179.409,6.060,149.264
C04622=1151.173,-33.192,-46.199,179.411,6.060,149.263
C04623=1151.168,-32.942,-46.211,179.414,6.061,149.263
C04624=1151.162,-32.693,-46.222,179.416,6.061,149.262
C04625=1151.157,-32.444,-46.235,179.418,6.062,149.261
C04626=1151.152,-32.194,-46.246,179.421,6.063,149.261
C04627=1151.147,-31.944,-46.258,179.423,6.063,149.260
C04628=1151.141,-31.694,-46.270,179.426,6.064,149.259
C04629=1151.136,-31.445,-46.282,179.428,6.065,149.259
C04630=1151.132,-31.195,-46.294,179.430,6.065,149.259
C04631=1151.126,-30.946,-46.306,179.432,6.065,149.258
C04632=1151.121,-30.696,-46.318,179.435,6.066,149.257
C04633=1151.116,-30.446,-46.330,179.437,6.066,149.257
C04634=1151.110,-30.196,-46.342,179.439,6.067,149.256
C04635=1151.105,-29.947,-46.353,179.442,6.067,149.256
C04636=1151.100,-29.697,-46.366,179.444,6.068,149.255
C04637=1151.095,-29.447,-46.378,179.447,6.069,149.254
C04638=1151.089,-29.197,-46.390,179.449,6.069,149.254
C04639=1151.084,-28.948,-46.402,179.452,6.070,149.253
C04640=1151.080,-28.699,-46.414,179.454,6.071,149.253
C04641=1151.074,-28.449,-46.425,179.456,6.071,149.252
C04642=1151.069,-28.199,-46.438,179.459,6.072,149.252
C04643=1151.064,-27.949,-46.450,179.461,6.073,149.251
C04644=1151.058,-27.699,-46.462,179.464,6.073,149.250
C04645=1151.054,-27.450,-46.474,179.466,6.074,149.250
C04646=1151.048,-27.200,-46.486,179.468,6.074,149.249
C04647=1151.043,-26.951,-46.498,179.471,6.075,149.249
C04648=1151.038,-26.701,-46.510,179.473,6.076,149.248
C04649=1151.032,-26.451,-46.522,179.476,6.076,149.248
C04650=1151.027,-26.202,-46.535,179.478,6.077,149.247
C04651=1151.022,-25.952,-46.547,179.480,6.078,149.246
C04652=1151.017,-25.703,-46.559,179.483,6.078,149.246
C04653=1151.012,-25.453,-46.570,179.485,6.079,149.245
C04654=1151.007,-25.203,-46.582,179.487,6.080,149.245
C04655=1151.002,-24.954,-46.595,179.490,6.080,149.244
C04656=1150.996,-24.683,-46.608,179.493,6.080,149.243
C04657=1150.990,-24.414,-46.622,179.495,6.081,149.243
C04658=1150.985,-24.144,-46.635,179.498,6.082,149.242
C04659=1150.979,-23.873,-46.648,179.501,6.083,149.241
C04660=1150.974,-23.624,-46.660,179.503,6.084,149.241
C04661=1150.969,-23.374,-46.672,179.505,6.084,149.241
C04662=1150.964,-23.125,-46.685,179.508,6.085,149.240
C04663=1150.958,-22.875,-46.697,179.510,6.086,149.239
C04664=1150.953,-22.626,-46.709,179.513,6.086,149.239
C04665=1150.948,-22.376,-46.721,179.515,6.087,149.238
C04666=1150.942,-22.126,-46.734,179.518,6.087,149.237
C04667=1150.937,-21.876,-46.746,179.520,6.088,149.237
C04668=1150.932,-21.627,-46.758,179.522,6.089,149.236
C04669=1150.927,-21.378,-46.771,179.525,6.089,149.236
C04670=1150.921,-21.128,-46.783,179.527,6.090,149.235
C04671=1150.917,-20.878,-46.796,179.529,6.091,149.235
C04672=1150.911,-20.628,-46.808,179.532,6.091,149.234
C04673=1150.906,-20.379,-46.820,179.534,6.092,149.234
C04674=1150.901,-20.129,-46.833,179.537,6.092,149.233
C04675=1150.896,-19.879,-46.845,179.539,6.093,149.232
C04676=1150.891,-19.630,-46.857,179.541,6.094,149.232
C04677=1150.885,-19.380,-46.869,179.544,6.094,149.231
C04678=1150.880,-19.131,-46.882,179.546,6.095,149.231
C04679=1150.875,-18.881,-46.894,179.549,6.095,149.230
C04680=1150.870,-18.631,-46.907,179.551,6.096,149.230
C04681=1150.865,-18.381,-46.919,179.554,6.097,149.229
C04682=1150.860,-18.132,-46.932,179.556,6.097,149.228
C04683=1150.854,-17.882,-46.944,179.558,6.098,149.228
C04684=1150.849,-17.633,-46.956,179.561,6.099,149.227
C04685=1150.844,-17.384,-46.969,179.563,6.099,149.227
C04686=1150.840,-17.134,-46.982,179.565,6.100,149.226
C04687=1150.833,-16.883,-46.994,179.568,6.100,149.225
C04688=1150.828,-16.634,-47.007,179.570,6.101,149.225
C04689=1150.823,-16.385,-47.020,179.572,6.102,149.224
C04690=1150.818,-16.135,-47.032,179.575,6.102,149.224
C04691=1150.813,-15.885,-47.044,179.577,6.103,149.223
C04692=1150.808,-15.635,-47.057,179.581,6.104,149.223
C04693=1150.803,-15.386,-47.070,179.583,6.105,149.222
C04694=1150.798,-15.137,-47.082,179.585,6.106,149.221
C04695=1150.792,-14.887,-47.094,179.588,6.106,149.221
C04696=1150.787,-14.637,-47.107,179.590,6.107,149.220
C04697=1150.782,-14.387,-47.120,179.592,6.108,149.220
C04698=1150.777,-14.138,-47.133,179.595,6.108,149.219
C04699=1150.772,-13.889,-47.145,179.597,6.109,149.219
C04700=1150.766,-13.639,-47.157,179.600,6.109,149.218
C04701=1150.761,-13.389,-47.170,179.602,6.110,149.217
C04702=1150.756,-13.139,-47.184,179.605,6.111,149.217
C04703=1150.751,-12.890,-47.196,179.607,6.111,149.216
C04704=1150.746,-12.640,-47.209,179.610,6.112,149.216
C04705=1150.741,-12.391,-47.221,179.612,6.113,149.215
C04706=1150.736,-12.141,-47.234,179.614,6.113,149.215
C04707=1150.731,-11.892,-47.247,179.617,6.114,149.214
C04708=1150.725,-11.641,-47.259,179.619,6.115,149.214
C04709=1150.720,-11.392,-47.272,179.622,6.116,149.213
C04710=1150.715,-11.142,-47.285,179.624,6.117,149.212
C04711=1150.710,-10.893,-47.298,179.627,6.117,149.212
C04712=1150.704,-10.643,-47.311,179.629,6.118,149.211
C04713=1150.699,-10.394,-47.323,179.632,6.118,149.211
C04714=1150.695,-10.144,-47.336,179.634,6.119,149.210
C04715=1150.689,-9.895,-47.349,179.637,6.120,149.209
C04716=1150.684,-9.645,-47.362,179.639,6.120,149.209
C04717=1150.679,-9.395,-47.375,179.641,6.121,149.208
C04718=1150.674,-9.146,-47.388,179.644,6.122,149.208
C04719=1150.669,-8.896,-47.400,179.646,6.122,149.207
C04720=1150.663,-8.647,-47.413,179.649,6.124,149.207
C04721=1150.658,-8.397,-47.426,179.651,6.125,149.206
C04722=1150.653,-8.147,-47.439,179.654,6.125,149.205
C04723=1150.648,-7.898,-47.452,179.656,6.126,149.205
C04724=1150.643,-7.648,-47.465,179.659,6.126,149.204
C04725=1150.638,-7.398,-47.478,179.661,6.127,149.204
C04726=1150.633,-7.149,-47.490,179.664,6.127,149.203
C04727=1150.627,-6.899,-47.504,179.666,6.128,149.203
C04728=1150.622,-6.649,-47.517,179.668,6.129,149.202
C04729=1150.617,-6.400,-47.529,179.671,6.129,149.201
C04730=1150.612,-6.150,-47.543,179.674,6.131,149.201
C04731=1150.607,-5.900,-47.555,179.676,6.132,149.200
C04732=1150.602,-5.651,-47.568,179.679,6.132,149.200
C04733=1150.597,-5.401,-47.582,179.681,6.133,149.199
C04734=1150.592,-5.152,-47.595,179.683,6.133,149.198
C04735=1150.586,-4.903,-47.607,179.686,6.134,149.198
C04736=1150.581,-4.652,-47.621,179.688,6.134,149.197
C04737=1150.576,-4.403,-47.634,179.690,6.135,149.197
C04738=1150.571,-4.153,-47.647,179.693,6.136,149.196
C04739=1150.566,-3.903,-47.660,179.696,6.137,149.196
C04740=1150.561,-3.655,-47.673,179.698,6.138,149.195
C04741=1150.556,-3.404,-47.687,179.701,6.139,149.195
C04742=1150.550,-3.155,-47.699,179.703,6.139,149.194
C04743=1150.545,-2.905,-47.712,179.706,6.140,149.193
C04744=1150.540,-2.655,-47.725,179.708,6.141,149.193
C04745=1150.535,-2.406,-47.738,179.710,6.141,149.192
C04746=1150.530,-2.156,-47.752,179.713,6.142,149.192
C04747=1150.525,-1.907,-47.765,179.716,6.143,149.191
C04748=1150.519,-1.657,-47.778,179.718,6.144,149.191
C04749=1150.515,-1.407,-47.791,179.721,6.144,149.190
C04750=1150.509,-1.158,-47.805,179.723,6.145,149.189
C04751=1150.504,-0.908,-47.818,179.725,6.146,149.189
C04752=1150.499,-0.659,-47.831,179.728,6.146,149.188
C04753=1150.493,-0.409,-47.844,179.730,6.147,149.188
C04754=1150.488,-0.160,-47.858,179.733,6.148,149.187
C04755=1150.483,0.090,-47.871,179.735,6.149,149.187
C04756=1150.478,0.340,-47.884,179.738,6.150,149.186
C04757=1150.473,0.589,-47.897,179.740,6.151,149.186
C04758=1150.468,0.839,-47.911,179.743,6.151,149.185
C04759=1150.463,1.088,-47.924,179.745,6.152,149.184
C04760=1150.457,1.358,-47.939,179.748,6.153,149.184
C04761=1150.452,1.628,-47.953,179.751,6.153,149.183
C04762=1150.446,1.896,-47.967,179.753,6.154,149.183
C04763=1150.441,2.166,-47.981,179.756,6.156,149.182
C04764=1150.435,2.415,-47.995,179.758,6.156,149.181
C04765=1150.431,2.665,-48.008,179.761,6.157,149.181
C04766=1150.425,2.914,-48.022,179.763,6.158,149.180
C04767=1150.421,3.164,-48.035,179.766,6.158,149.180
C04768=1150.415,3.414,-48.048,179.768,6.159,149.179
C04769=1150.410,3.663,-48.062,179.771,6.160,149.178
C04770=1150.405,3.913,-48.075,179.773,6.161,149.178
C04771=1150.400,4.163,-48.089,179.776,6.161,149.177
C04772=1150.395,4.412,-48.102,179.778,6.162,149.177
C04773=1150.389,4.662,-48.115,179.781,6.163,149.176
C04774=1150.384,4.911,-48.129,179.783,6.163,149.176
C04775=1150.379,5.161,-48.142,179.786,6.165,149.175
C04776=1150.374,5.410,-48.156,179.789,6.165,149.174
C04777=1150.369,5.660,-48.169,179.791,6.166,149.174
C04778=1150.364,5.910,-48.183,179.793,6.167,149.173
C04779=1150.359,6.159,-48.196,179.796,6.168,149.173
C04780=1150.354,6.409,-48.210,179.799,6.169,149.172
C04781=1150.348,6.659,-48.224,179.801,6.170,149.172
C04782=1150.344,6.908,-48.237,179.804,6.170,149.171
C04783=1150.338,7.158,-48.250,179.806,6.171,149.171
C04784=1150.333,7.407,-48.265,179.808,6.171,149.170
C04785=1150.328,7.656,-48.278,179.811,6.173,149.169
C04786=1150.323,7.906,-48.292,179.814,6.173,149.169
C04787=1150.318,8.156,-48.306,179.816,6.174,149.168
C04788=1150.313,8.405,-48.318,179.819,6.175,149.168
C04789=1150.308,8.655,-48.333,179.821,6.175,149.167
C04790=1150.302,8.905,-48.346,179.824,6.177,149.166
C04791=1150.298,9.154,-48.360,179.826,6.178,149.166
C04792=1150.292,9.403,-48.374,179.828,6.178,149.166
C04793=1150.287,9.654,-48.387,179.831,6.179,149.165
C04794=1150.282,9.903,-48.401,179.833,6.180,149.164
C04795=1150.277,10.152,-48.415,179.837,6.181,149.164
C04796=1150.272,10.402,-48.428,179.839,6.182,149.163
C04797=1150.267,10.651,-48.442,179.841,6.182,149.163
C04798=1150.262,10.901,-48.456,179.844,6.183,149.162
C04799=1150.257,11.151,-48.469,179.846,6.183,149.161
C04800=1150.252,11.400,-48.483,179.849,6.185,149.161
C04801=1150.247,11.650,-48.498,179.852,6.185,149.160
C04802=1150.241,11.900,-48.511,179.854,6.186,149.160
C04803=1150.236,12.149,-48.525,179.856,6.187,149.159
C04804=1150.232,12.398,-48.539,179.859,6.188,149.159
C04805=1150.226,12.648,-48.552,179.861,6.189,149.158
C04806=1150.221,12.898,-48.566,179.864,6.190,149.158
C04807=1150.216,13.147,-48.581,179.866,6.190,149.157
C04808=1150.210,13.396,-48.594,179.869,6.191,149.156
C04809=1150.206,13.647,-48.607,179.872,6.193,149.156
C04810=1150.201,13.896,-48.622,179.874,6.193,149.155
C04811=1150.195,14.145,-48.636,179.876,6.194,149.155
C04812=1150.190,14.395,-48.650,179.879,6.194,149.154
C04813=1150.185,14.645,-48.664,179.882,6.196,149.154
C04814=1150.179,14.894,-48.677,179.885,6.196,149.153
C04815=1150.175,15.144,-48.691,179.887,6.197,149.152
C04816=1150.170,15.393,-48.705,179.889,6.198,149.152
C04817=1150.165,15.642,-48.719,179.892,6.199,149.151
C04818=1150.160,15.892,-48.733,179.894,6.200,149.151
C04819=1150.155,16.142,-48.748,179.897,6.200,149.150
C04820=1150.150,16.392,-48.761,179.899,6.201,149.150
C04821=1150.144,16.641,-48.775,179.902,6.203,149.149
C04822=1150.139,16.891,-48.789,179.905,6.203,149.149
C04823=1150.135,17.140,-48.803,179.907,6.204,149.148
C04824=1150.129,17.389,-48.817,179.909,6.205,149.147
C04825=1150.124,17.639,-48.831,179.913,6.206,149.147
C04826=1150.119,17.889,-48.846,179.915,6.207,149.146
C04827=1150.114,18.138,-48.860,179.917,6.207,149.146
C04828=1150.109,18.387,-48.874,179.920,6.208,149.145
C04829=1150.104,18.638,-48.887,179.922,6.210,149.145
C04830=1150.099,18.887,-48.902,179.925,6.210,149.144
C04831=1150.094,19.137,-48.916,179.927,6.211,149.144
C04832=1150.088,19.386,-48.930,179.930,6.211,149.143
C04833=1150.083,19.636,-48.944,179.933,6.213,149.142
C04834=1150.078,19.886,-48.958,179.935,6.213,149.142
C04835=1150.073,20.135,-48.973,179.937,6.214,149.141
C04836=1150.068,20.384,-48.987,179.940,6.215,149.141
C04837=1150.063,20.634,-49.001,179.943,6.216,149.140
C04838=1150.058,20.884,-49.015,179.945,6.217,149.139
C04839=1150.053,21.133,-49.029,179.948,6.218,149.139
C04840=1150.047,21.382,-49.043,179.950,6.219,149.139
C04841=1150.042,21.632,-49.058,179.953,6.220,149.138
C04842=1150.037,21.882,-49.072,179.955,6.221,149.137
C04843=1150.033,22.131,-49.087,179.958,6.221,149.137
C04844=1150.028,22.381,-49.101,179.961,6.223,149.136
C04845=1150.022,22.630,-49.115,179.963,6.223,149.136
C04846=1150.017,22.879,-49.129,179.965,6.224,149.135
C04847=1150.012,23.129,-49.144,179.969,6.225,149.134
C04848=1150.007,23.379,-49.158,179.971,6.226,149.134
C04849=1150.002,23.629,-49.172,179.973,6.227,149.134
C04850=1149.997,23.878,-49.186,179.976,6.227,149.133
C04851=1149.992,24.127,-49.200,179.978,6.229,149.132
C04852=1149.987,24.376,-49.215,179.981,6.229,149.132
C04853=1149.982,24.626,-49.230,179.983,6.230,149.131
C04854=1149.977,24.876,-49.245,179.986,6.231,149.131
C04855=1149.972,25.126,-49.259,179.989,6.232,149.130
C04856=1149.967,25.376,-49.273,179.991,6.233,149.129
C04857=1149.962,25.625,-49.287,179.994,6.234,149.129
C04858=1149.956,25.874,-49.302,179.997,6.235,149.128
C04859=1149.951,26.123,-49.316,179.999,6.236,149.128
C04860=1149.947,26.373,-49.331,-179.998,6.237,149.127
C04861=1149.941,26.623,-49.345,-179.996,6.238,149.127
C04862=1149.936,26.873,-49.360,-179.994,6.239,149.126
C04863=1149.931,27.122,-49.375,-179.991,6.239,149.126
C04864=1149.926,27.391,-49.390,-179.988,6.241,149.125
C04865=1149.921,27.660,-49.405,-179.986,6.241,149.125
C04866=1149.914,27.928,-49.421,-179.982,6.242,149.124
C04867=1149.909,28.197,-49.437,-179.980,6.243,149.123
C04868=1149.904,28.447,-49.451,-179.977,6.244,149.123
C04869=1149.899,28.697,-49.466,-179.975,6.245,149.122
C04870=1149.894,28.946,-49.481,-179.972,6.246,149.122
C04871=1149.889,29.196,-49.495,-179.969,6.247,149.121
C04872=1149.884,29.445,-49.510,-179.967,6.248,149.121
C04873=1149.879,29.695,-49.525,-179.964,6.249,149.120
C04874=1149.874,29.944,-49.539,-179.962,6.250,149.120
C04875=1149.869,30.194,-49.554,-179.959,6.251,149.119
C04876=1149.864,30.443,-49.569,-179.957,6.252,149.118
C04877=1149.859,30.693,-49.583,-179.954,6.253,149.118
C04878=1149.854,30.942,-49.598,-179.952,6.254,149.117
C04879=1149.848,31.192,-49.613,-179.948,6.255,149.117
C04880=1149.843,31.441,-49.627,-179.946,6.256,149.116
C04881=1149.838,31.690,-49.642,-179.944,6.257,149.116
C04882=1149.833,31.940,-49.657,-179.941,6.258,149.115
C04883=1149.828,32.189,-49.672,-179.939,6.259,149.115
C04884=1149.823,32.439,-49.686,-179.936,6.259,149.114
C04885=1149.818,32.689,-49.700,-179.933,6.261,149.113
C04886=1149.813,32.938,-49.716,-179.930,6.261,149.113
C04887=1149.808,33.188,-49.730,-179.928,6.262,149.112
C04888=1149.803,33.437,-49.745,-179.926,6.264,149.112
C04889=1149.797,33.687,-49.760,-179.923,6.264,149.111
C04890=1149.793,33.936,-49.775,-179.921,6.265,149.111
C04891=1149.788,34.186,-49.789,-179.918,6.266,149.110
C04892=1149.783,34.435,-49.805,-179.915,6.267,149.110
C04893=1149.778,34.685,-49.819,-179.912,6.268,149.109
C04894=1149.773,34.934,-49.834,-179.910,6.269,149.108
C04895=1149.767,35.184,-49.849,-179.908,6.270,149.108
C04896=1149.763,35.433,-49.864,-179.905,6.271,149.107
C04897=1149.757,35.683,-49.880,-179.902,6.272,149.107
C04898=1149.752,35.932,-49.894,-179.900,6.273,149.106
C04899=1149.748,36.181,-49.909,-179.897,6.274,149.106
C04900=1149.742,36.431,-49.924,-179.894,6.275,149.105
C04901=1149.737,36.681,-49.939,-179.892,6.276,149.105
C04902=1149.732,36.931,-49.954,-179.889,6.277,149.104
C04903=1149.727,37.180,-49.969,-179.887,6.278,149.104
C04904=1149.723,37.429,-49.984,-179.884,6.279,149.103
C04905=1149.717,37.679,-49.999,-179.881,6.280,149.102
C04906=1149.712,37.929,-50.014,-179.879,6.281,149.102
C04907=1149.707,38.178,-50.029,-179.876,6.282,149.101
C04908=1149.702,38.428,-50.044,-179.874,6.283,149.101
C04909=1149.697,38.677,-50.059,-179.871,6.284,149.100
C04910=1149.692,38.926,-50.074,-179.868,6.285,149.100
C04911=1149.686,39.176,-50.089,-179.866,6.286,149.099
C04912=1149.682,39.425,-50.104,-179.863,6.287,149.099
C04913=1149.676,39.675,-50.120,-179.861,6.288,149.098
C04914=1149.671,39.924,-50.134,-179.858,6.290,149.098
C04915=1149.667,40.174,-50.150,-179.855,6.290,149.097
C04916=1149.662,40.424,-50.165,-179.853,6.291,149.097
C04917=1149.657,40.673,-50.181,-179.850,6.292,149.096
C04918=1149.652,40.923,-50.195,-179.848,6.293,149.095
C04919=1149.646,41.172,-50.210,-179.845,6.294,149.095
C04920=1149.642,41.421,-50.225,-179.842,6.295,149.094
C04921=1149.636,41.671,-50.241,-179.840,6.297,149.094
C04922=1149.631,41.920,-50.255,-179.837,6.297,149.093
C04923=1149.626,42.170,-50.271,-179.835,6.298,149.093
C04924=1149.622,42.419,-50.286,-179.832,6.299,149.092
C04925=1149.616,42.669,-50.302,-179.830,6.300,149.092
C04926=1149.611,42.918,-50.317,-179.827,6.302,149.091
C04927=1149.606,43.167,-50.332,-179.824,6.302,149.091
C04928=1149.601,43.417,-50.347,-179.822,6.303,149.090
C04929=1149.596,43.666,-50.362,-179.819,6.304,149.089
C04930=1149.591,43.917,-50.378,-179.817,6.305,149.089
C04931=1149.587,44.166,-50.393,-179.813,6.306,149.088
C04932=1149.581,44.415,-50.409,-179.811,6.307,149.088
C04933=1149.576,44.664,-50.424,-179.808,6.309,149.087
C04934=1149.571,44.914,-50.439,-179.806,6.309,149.087
C04935=1149.566,45.164,-50.455,-179.803,6.311,149.086
C04936=1149.561,45.413,-50.471,-179.800,6.312,149.086
C04937=1149.556,45.663,-50.485,-179.798,6.312,149.085
C04938=1149.551,45.912,-50.501,-179.795,6.314,149.085
C04939=1149.546,46.161,-50.516,-179.793,6.315,149.084
C04940=1149.541,46.411,-50.532,-179.790,6.316,149.084
C04941=1149.536,46.661,-50.547,-179.787,6.317,149.083
C04942=1149.531,46.910,-50.562,-179.785,6.318,149.082
C04943=1149.526,47.159,-50.578,-179.783,6.319,149.082
C04944=1149.521,47.409,-50.594,-179.779,6.320,149.081
C04945=1149.516,47.659,-50.609,-179.777,6.321,149.081
C04946=1149.511,47.908,-50.624,-179.774,6.322,149.080
C04947=1149.506,48.157,-50.640,-179.772,6.323,149.080
C04948=1149.501,48.407,-50.656,-179.770,6.324,149.079
C04949=1149.496,48.656,-50.671,-179.766,6.326,149.079
C04950=1149.491,48.906,-50.687,-179.764,6.326,149.078
C04951=1149.486,49.155,-50.703,-179.761,6.328,149.078
C04952=1149.482,49.404,-50.718,-179.759,6.328,149.077
C04953=1149.476,49.654,-50.734,-179.756,6.330,149.077
C04954=1149.471,49.903,-50.749,-179.753,6.331,149.076
C04955=1149.466,50.153,-50.765,-179.751,6.332,149.076
C04956=1149.461,50.402,-50.780,-179.748,6.333,149.075
C04957=1149.456,50.652,-50.796,-179.745,6.334,149.074
C04958=1149.451,50.901,-50.812,-179.743,6.335,149.074
C04959=1149.446,51.151,-50.827,-179.740,6.337,149.073
C04960=1149.441,51.400,-50.844,-179.738,6.337,149.073
C04961=1149.436,51.649,-50.859,-179.734,6.339,149.072
C04962=1149.431,51.899,-50.875,-179.732,6.339,149.072
C04963=1149.426,52.149,-50.890,-179.730,6.341,149.071
C04964=1149.421,52.398,-50.906,-179.727,6.342,149.071
C04965=1149.416,52.648,-50.922,-179.725,6.342,149.070
C04966=1149.412,52.897,-50.938,-179.722,6.344,149.070
C04967=1149.406,53.146,-50.953,-179.719,6.345,149.069
C04968=1149.401,53.415,-50.970,-179.717,6.346,149.069
C04969=1149.396,53.684,-50.988,-179.713,6.348,149.068
C04970=1149.390,53.952,-51.005,-179.710,6.349,149.067
C04971=1149.384,54.221,-51.022,-179.708,6.350,149.067
C04972=1149.379,54.470,-51.037,-179.705,6.351,149.067
C04973=1149.374,54.720,-51.053,-179.703,6.352,149.066
C04974=1149.369,54.969,-51.069,-179.700,6.353,149.065
C04975=1149.364,55.218,-51.085,-179.697,6.354,149.065
C04976=1149.360,55.468,-51.100,-179.694,6.356,149.064
C04977=1149.355,55.717,-51.117,-179.692,6.356,149.064
C04978=1149.350,55.967,-51.133,-179.689,6.358,149.063
C04979=1149.345,56.217,-51.148,-179.687,6.359,149.063
C04980=1149.339,56.465,-51.165,-179.684,6.360,149.062
C04981=1149.335,56.715,-51.180,-179.682,6.361,149.062
C04982=1149.329,56.965,-51.196,-179.679,6.362,149.061
C04983=1149.325,57.214,-51.213,-179.676,6.363,149.061
C04984=1149.319,57.464,-51.228,-179.673,6.364,149.060
C04985=1149.314,57.713,-51.244,-179.671,6.365,149.060
C04986=1149.310,57.963,-51.261,-179.668,6.367,149.059
C04987=1149.304,58.212,-51.276,-179.666,6.367,149.059
C04988=1149.300,58.461,-51.293,-179.663,6.369,149.058
C04989=1149.294,58.711,-51.308,-179.660,6.370,149.057
C04990=1149.289,58.960,-51.325,-179.658,6.371,149.057
C04991=1149.284,59.210,-51.341,-179.655,6.373,149.056
C04992=1149.279,59.459,-51.356,-179.652,6.373,149.056
C04993=1149.275,59.709,-51.373,-179.650,6.375,149.055
C04994=1149.269,59.958,-51.389,-179.647,6.376,149.055
C04995=1149.265,60.208,-51.405,-179.644,6.377,149.054
C04996=1149.259,60.457,-51.421,-179.642,6.378,149.054
C04997=1149.255,60.706,-51.437,-179.639,6.379,149.053
C04998=1149.249,60.956,-51.453,-179.637,6.380,149.053
C04999=1149.245,61.205,-51.470,-179.633,6.381,149.052
C05000=1149.240,61.455,-51.485,-179.631,6.383,149.052
C05001=1149.235,61.704,-51.502,-179.629,6.384,149.051
C05002=1149.230,61.953,-51.518,-179.625,6.385,149.051
C05003=1149.225,62.203,-51.534,-179.623,6.386,149.050
C05004=1149.219,62.452,-51.551,-179.620,6.388,149.050
C05005=1149.215,62.702,-51.567,-179.618,6.388,149.049
C05006=1149.210,62.951,-51.583,-179.615,6.390,149.049
C05007=1149.205,63.201,-51.600,-179.613,6.391,149.048
C05008=1149.200,63.450,-51.616,-179.610,6.392,149.048
C05009=1149.195,63.699,-51.632,-179.607,6.394,149.047
C05010=1149.190,63.949,-51.648,-179.605,6.395,149.047
C05011=1149.185,64.198,-51.665,-179.602,6.396,149.046
C05012=1149.180,64.447,-51.681,-179.599,6.397,149.046
C05013=1149.175,64.698,-51.697,-179.597,6.398,149.045
C05014=1149.170,64.946,-51.714,-179.594,6.399,149.044
C05015=1149.165,65.196,-51.730,-179.591,6.401,149.044
C05016=1149.160,65.445,-51.747,-179.588,6.402,149.043
C05017=1149.155,65.695,-51.763,-179.586,6.403,149.043
C05018=1149.151,65.944,-51.779,-179.583,6.404,149.043
C05019=1149.145,66.193,-51.796,-179.581,6.405,149.042
C05020=1149.140,66.443,-51.812,-179.578,6.407,149.041
C05021=1149.135,66.692,-51.828,-179.576,6.407,149.041
C05022=1149.131,66.942,-51.845,-179.572,6.409,149.040
C05023=1149.126,67.191,-51.862,-179.570,6.410,149.040
C05024=1149.120,67.441,-51.878,-179.567,6.411,149.039
C05025=1149.116,67.690,-51.895,-179.564,6.413,149.039
C05026=1149.110,67.939,-51.911,-179.562,6.413,149.038
C05027=1149.106,68.189,-51.928,-179.559,6.415,149.038
C05028=1149.101,68.438,-51.945,-179.556,6.416,149.037
C05029=1149.096,68.687,-51.961,-179.554,6.417,149.037
C05030=1149.091,68.937,-51.977,-179.551,6.419,149.036
C05031=1149.086,69.186,-51.993,-179.549,6.419,149.036
C05032=1149.081,69.436,-52.011,-179.546,6.421,149.035
C05033=1149.076,69.685,-52.027,-179.543,6.423,149.035
C05034=1149.071,69.934,-52.044,-179.540,6.423,149.034
C05035=1149.066,70.184,-52.061,-179.538,6.425,149.034
C05036=1149.061,70.433,-52.078,-179.535,6.426,149.033
C05037=1149.056,70.683,-52.093,-179.532,6.427,149.033
C05038=1149.051,70.933,-52.110,-179.530,6.429,149.032
C05039=1149.046,71.182,-52.127,-179.527,6.430,149.032
C05040=1149.041,71.431,-52.143,-179.524,6.431,149.031
C05041=1149.036,71.681,-52.161,-179.522,6.432,149.031
C05042=1149.032,71.930,-52.177,-179.519,6.433,149.030
C05043=1149.026,72.179,-52.194,-179.516,6.435,149.030
C05044=1149.021,72.429,-52.211,-179.513,6.436,149.029
C05045=1149.017,72.678,-52.228,-179.511,6.437,149.029
C05046=1149.012,72.927,-52.244,-179.508,6.438,149.028
C05047=1149.006,73.177,-52.261,-179.506,6.439,149.028
C05048=1149.002,73.426,-52.278,-179.503,6.441,149.027
C05049=1148.996,73.675,-52.295,-179.500,6.443,149.027
C05050=1148.992,73.925,-52.311,-179.498,6.443,149.026
C05051=1148.987,74.174,-52.328,-179.495,6.445,149.026
C05052=1148.982,74.424,-52.345,-179.492,6.446,149.025
C05053=1148.977,74.673,-52.362,-179.490,6.447,149.025
C05054=1148.972,74.923,-52.379,-179.487,6.449,149.024
C05055=1148.967,75.172,-52.396,-179.484,6.450,149.024
C05056=1148.962,75.421,-52.413,-179.482,6.451,149.023
C05057=1148.957,75.670,-52.430,-179.479,6.452,149.023
C05058=1148.953,75.920,-52.447,-179.476,6.454,149.022
C05059=1148.947,76.169,-52.464,-179.473,6.455,149.022
C05060=1148.942,76.418,-52.480,-179.471,6.456,149.021
C05061=1148.937,76.668,-52.497,-179.469,6.457,149.021
C05062=1148.933,76.917,-52.514,-179.465,6.458,149.020
C05063=1148.928,77.167,-52.532,-179.463,6.460,149.020
C05064=1148.923,77.416,-52.549,-179.460,6.461,149.019
C05065=1148.917,77.665,-52.566,-179.458,6.463,149.019
C05066=1148.913,77.915,-52.582,-179.454,6.464,149.018
C05067=1148.908,78.165,-52.600,-179.452,6.465,149.018
C05068=1148.904,78.413,-52.617,-179.450,6.467,149.017
C05069=1148.898,78.662,-52.634,-179.446,6.468,149.017
C05070=1148.893,78.912,-52.651,-179.444,6.469,149.016
C05071=1148.888,79.162,-52.668,-179.441,6.470,149.016
C05072=1148.883,79.431,-52.686,-179.438,6.472,149.015
C05073=1148.878,79.698,-52.705,-179.435,6.473,149.015
C05074=1148.872,79.967,-52.724,-179.432,6.475,149.014
C05075=1148.867,80.236,-52.742,-179.430,6.476,149.014
C05076=1148.862,80.484,-52.759,-179.427,6.477,149.013
C05077=1148.857,80.734,-52.776,-179.424,6.478,149.013
C05078=1148.853,80.983,-52.793,-179.421,6.480,149.012
C05079=1148.847,81.233,-52.810,-179.419,6.481,149.012
C05080=1148.842,81.483,-52.828,-179.416,6.482,149.011
C05081=1148.838,81.731,-52.845,-179.413,6.484,149.011
C05082=1148.832,81.981,-52.862,-179.411,6.486,149.010
C05083=1148.827,82.230,-52.880,-179.408,6.487,149.010
C05084=1148.823,82.479,-52.897,-179.405,6.488,149.009
C05085=1148.817,82.729,-52.914,-179.402,6.490,149.009
C05086=1148.813,82.978,-52.932,-179.400,6.490,149.008
C05087=1148.808,83.228,-52.949,-179.398,6.492,149.008
C05088=1148.803,83.477,-52.967,-179.394,6.493,149.007
C05089=1148.798,83.727,-52.984,-179.392,6.494,149.007
C05090=1148.793,83.975,-53.000,-179.389,6.496,149.006
C05091=1148.788,84.225,-53.018,-179.386,6.497,149.006
C05092=1148.783,84.474,-53.035,-179.384,6.499,149.005
C05093=1148.779,84.723,-53.053,-179.381,6.500,149.005
C05094=1148.773,84.973,-53.070,-179.379,6.501,149.004
C05095=1148.768,85.222,-53.088,-179.375,6.503,149.004
C05096=1148.763,85.472,-53.105,-179.373,6.504,149.003
C05097=1148.759,85.721,-53.123,-179.371,6.505,149.003
C05098=1148.754,85.971,-53.140,-179.368,6.507,149.003
C05099=1148.749,86.220,-53.158,-179.365,6.508,149.002
C05100=1148.744,86.470,-53.175,-179.362,6.509,149.001
C05101=1148.740,86.719,-53.193,-179.360,6.511,149.001
C05102=1148.735,86.968,-53.211,-179.357,6.512,149.000
C05103=1148.729,87.218,-53.228,-179.354,6.514,149.000
C05104=1148.724,87.466,-53.245,-179.352,6.515,149.000
C05105=1148.719,87.715,-53.262,-179.349,6.516,148.999
C05106=1148.714,87.965,-53.280,-179.346,6.518,148.998
C05107=1148.710,88.214,-53.298,-179.343,6.519,148.998
C05108=1148.704,88.464,-53.315,-179.341,6.520,148.998
C05109=1148.699,88.713,-53.333,-179.338,6.522,148.997
C05110=1148.695,88.962,-53.351,-179.335,6.523,148.997
C05111=1148.690,89.211,-53.368,-179.332,6.525,148.996
C05112=1148.685,89.461,-53.386,-179.330,6.526,148.996
C05113=1148.680,89.710,-53.404,-179.327,6.527,148.995
C05114=1148.675,89.960,-53.421,-179.324,6.529,148.995
C05115=1148.670,90.209,-53.439,-179.321,6.530,148.994
C05116=1148.665,90.458,-53.457,-179.319,6.531,148.994
C05117=1148.660,90.708,-53.474,-179.316,6.533,148.993
C05118=1148.656,90.957,-53.492,-179.313,6.534,148.993
C05119=1148.651,91.206,-53.510,-179.310,6.536,148.992
C05120=1148.646,91.455,-53.528,-179.308,6.537,148.992
C05121=1148.641,91.705,-53.545,-179.306,6.539,148.991
C05122=1148.636,91.955,-53.563,-179.302,6.540,148.991
C05123=1148.632,92.204,-53.581,-179.300,6.542,148.990
C05124=1148.627,92.453,-53.599,-179.297,6.542,148.990
C05125=1148.622,92.702,-53.617,-179.295,6.544,148.990
C05126=1148.616,92.952,-53.635,-179.292,6.546,148.989
C05127=1148.612,93.201,-53.653,-179.289,6.547,148.989
C05128=1148.607,93.450,-53.671,-179.286,6.549,148.988
C05129=1148.602,93.699,-53.688,-179.284,6.550,148.988
C05130=1148.597,93.949,-53.706,-179.281,6.551,148.987
C05131=1148.592,94.198,-53.724,-179.278,6.553,148.987
C05132=1148.587,94.447,-53.742,-179.275,6.554,148.986
C05133=1148.582,94.697,-53.760,-179.273,6.556,148.986
C05134=1148.577,94.946,-53.778,-179.270,6.557,148.985
C05135=1148.573,95.196,-53.796,-179.267,6.558,148.985
C05136=1148.568,95.445,-53.814,-179.264,6.560,148.984
C05137=1148.563,95.694,-53.832,-179.262,6.562,148.984
C05138=1148.558,95.943,-53.850,-179.259,6.563,148.983
C05139=1148.553,96.193,-53.868,-179.257,6.564,148.983
C05140=1148.548,96.442,-53.886,-179.254,6.565,148.982
C05141=1148.543,96.691,-53.904,-179.251,6.567,148.982
C05142=1148.538,96.940,-53.922,-179.248,6.569,148.982
C05143=1148.534,97.190,-53.940,-179.245,6.570,148.981
C05144=1148.529,97.439,-53.958,-179.243,6.571,148.981
C05145=1148.524,97.688,-53.976,-179.240,6.573,148.980
C05146=1148.519,97.937,-53.994,-179.237,6.574,148.980
C05147=1148.514,98.187,-54.012,-179.235,6.576,148.979
C05148=1148.509,98.436,-54.030,-179.232,6.578,148.979
C05149=1148.504,98.686,-54.049,-179.229,6.578,148.978
C05150=1148.499,98.935,-54.067,-179.227,6.580,148.978
C05151=1148.494,99.184,-54.085,-179.224,6.582,148.977
C05152=1148.490,99.434,-54.103,-179.221,6.583,148.977
C05153=1148.485,99.683,-54.121,-179.218,6.585,148.977
C05154=1148.480,99.931,-54.140,-179.215,6.586,148.976
C05155=1148.476,100.181,-54.158,-179.213,6.587,148.975
C05156=1148.471,100.430,-54.176,-179.210,6.589,148.975
C05157=1148.465,100.680,-54.195,-179.208,6.591,148.975
C05158=1148.460,100.929,-54.213,-179.205,6.592,148.974
C05159=1148.455,101.178,-54.231,-179.202,6.594,148.974
C05160=1148.451,101.428,-54.249,-179.199,6.595,148.973
C05161=1148.446,101.677,-54.268,-179.197,6.596,148.973
C05162=1148.441,101.926,-54.286,-179.194,6.598,148.972
C05163=1148.436,102.175,-54.304,-179.191,6.600,148.972
C05164=1148.432,102.425,-54.322,-179.188,6.601,148.971
C05165=1148.427,102.674,-54.340,-179.185,6.603,148.971
C05166=1148.421,102.923,-54.360,-179.183,6.604,148.970
C05167=1148.416,103.172,-54.378,-179.180,6.605,148.970
C05168=1148.412,103.422,-54.396,-179.178,6.607,148.970
C05169=1148.407,103.671,-54.415,-179.175,6.608,148.969
C05170=1148.402,103.920,-54.433,-179.172,6.610,148.969
C05171=1148.397,104.169,-54.451,-179.169,6.611,148.968
C05172=1148.393,104.419,-54.470,-179.166,6.613,148.968
C05173=1148.388,104.668,-54.488,-179.164,6.615,148.967
C05174=1148.382,104.917,-54.507,-179.161,6.616,148.967
C05175=1148.378,105.167,-54.525,-179.159,6.617,148.967
C05176=1148.373,105.435,-54.545,-179.156,6.619,148.966
C05177=1148.367,105.703,-54.565,-179.152,6.621,148.966
C05178=1148.362,105.972,-54.585,-179.149,6.623,148.965
C05179=1148.357,106.240,-54.605,-179.146,6.624,148.964
C05180=1148.353,106.490,-54.624,-179.144,6.626,148.964
C05181=1148.347,106.739,-54.642,-179.141,6.627,148.964
C05182=1148.342,106.988,-54.661,-179.139,6.629,148.963
C05183=1148.338,107.237,-54.679,-179.136,6.630,148.963
C05184=1148.333,107.486,-54.699,-179.133,6.632,148.962
C05185=1148.328,107.736,-54.717,-179.130,6.633,148.962
C05186=1148.323,107.985,-54.735,-179.127,6.635,148.961
C05187=1148.318,108.234,-54.754,-179.125,6.637,148.961
C05188=1148.313,108.483,-54.772,-179.122,6.638,148.961
C05189=1148.308,108.733,-54.792,-179.119,6.640,148.960
C05190=1148.303,108.982,-54.810,-179.116,6.641,148.959
C05191=1148.299,109.231,-54.829,-179.114,6.642,148.959
C05192=1148.294,109.481,-54.848,-179.111,6.644,148.959
C05193=1148.289,109.729,-54.866,-179.108,6.646,148.958
C05194=1148.284,109.980,-54.885,-179.106,6.647,148.958
C05195=1148.280,110.228,-54.904,-179.103,6.649,148.957
C05196=1148.275,110.478,-54.924,-179.100,6.651,148.957
C05197=1148.270,110.727,-54.942,-179.097,6.652,148.956
C05198=1148.265,110.976,-54.961,-179.094,6.654,148.956
C05199=1148.260,111.226,-54.979,-179.091,6.655,148.956
C05200=1148.255,111.475,-54.999,-179.089,6.657,148.955
C05201=1148.251,111.724,-55.018,-179.087,6.658,148.955
C05202=1148.245,111.973,-55.036,-179.084,6.660,148.954
C05203=1148.241,112.222,-55.055,-179.081,6.661,148.954
C05204=1148.236,112.472,-55.074,-179.078,6.663,148.953
C05205=1148.231,112.721,-55.093,-179.075,6.664,148.953
C05206=1148.226,112.970,-55.112,-179.072,6.666,148.953
C05207=1148.221,113.219,-55.130,-179.070,6.668,148.952
C05208=1148.217,113.469,-55.150,-179.067,6.669,148.952
C05209=1148.212,113.717,-55.169,-179.064,6.671,148.951
C05210=1148.207,113.967,-55.188,-179.062,6.673,148.951
C05211=1148.202,114.217,-55.207,-179.059,6.675,148.950
C05212=1148.197,114.465,-55.225,-179.056,6.676,148.950
C05213=1148.192,114.715,-55.245,-179.053,6.678,148.949
C05214=1148.188,114.963,-55.264,-179.050,6.679,148.949
C05215=1148.183,115.213,-55.283,-179.048,6.680,148.949
C05216=1148.178,115.462,-55.301,-179.045,6.682,148.948
C05217=1148.173,115.712,-55.321,-179.043,6.684,148.948
C05218=1148.168,115.960,-55.340,-179.040,6.685,148.947
C05219=1148.164,116.210,-55.359,-179.037,6.687,148.947
C05220=1148.158,116.459,-55.378,-179.034,6.688,148.946
C05221=1148.153,116.709,-55.398,-179.031,6.690,148.946
C05222=1148.149,116.957,-55.416,-179.029,6.692,148.946
C05223=1148.144,117.207,-55.436,-179.026,6.693,148.945
C05224=1148.139,117.456,-55.455,-179.023,6.695,148.945
C05225=1148.135,117.705,-55.474,-179.020,6.697,148.944
C05226=1148.130,117.955,-55.494,-179.018,6.698,148.944
C05227=1148.124,118.204,-55.513,-179.015,6.700,148.944
C05228=1148.120,118.453,-55.532,-179.012,6.702,148.943
C05229=1148.115,118.702,-55.551,-179.009,6.704,148.943
C05230=1148.110,118.952,-55.571,-179.006,6.705,148.942
C05231=1148.105,119.201,-55.590,-179.004,6.707,148.942
C05232=1148.101,119.450,-55.609,-179.001,6.708,148.941
C05233=1148.096,119.699,-55.628,-178.998,6.710,148.941
C05234=1148.091,119.948,-55.648,-178.995,6.712,148.941
C05235=1148.087,120.198,-55.667,-178.993,6.713,148.940
C05236=1148.082,120.446,-55.686,-178.990,6.715,148.940
C05237=1148.077,120.696,-55.706,-178.987,6.717,148.939
C05238=1148.071,120.945,-55.725,-178.985,6.719,148.939
C05239=1148.067,121.194,-55.745,-178.982,6.720,148.939
C05240=1148.063,121.444,-55.764,-178.979,6.722,148.938
C05241=1148.057,121.693,-55.783,-178.976,6.724,148.938
C05242=1148.053,121.942,-55.803,-178.973,6.725,148.937
C05243=1148.047,122.191,-55.822,-178.970,6.727,148.937
C05244=1148.043,122.441,-55.842,-178.968,6.728,148.936
C05245=1148.039,122.689,-55.862,-178.965,6.730,148.936
C05246=1148.033,122.938,-55.881,-178.962,6.732,148.935
C05247=1148.029,123.188,-55.901,-178.960,6.733,148.935
C05248=1148.024,123.437,-55.920,-178.957,6.735,148.935
C05249=1148.019,123.686,-55.939,-178.954,6.737,148.934
C05250=1148.014,123.936,-55.959,-178.951,6.739,148.934
C05251=1148.010,124.185,-55.978,-178.949,6.740,148.933
C05252=1148.005,124.433,-55.998,-178.946,6.742,148.933
C05253=1148.000,124.683,-56.018,-178.943,6.744,148.933
C05254=1147.995,124.932,-56.038,-178.941,6.745,148.932
C05255=1147.990,125.181,-56.057,-178.938,6.747,148.932
C05256=1147.985,125.431,-56.076,-178.935,6.749,148.931
C05257=1147.981,125.680,-56.097,-178.932,6.750,148.931
C05258=1147.975,125.928,-56.116,-178.929,6.752,148.930
C05259=1147.971,126.178,-56.136,-178.926,6.754,148.930
C05260=1147.967,126.427,-56.155,-178.924,6.755,148.930
C05261=1147.962,126.676,-56.175,-178.921,6.757,148.929
C05262=1147.957,126.925,-56.195,-178.918,6.759,148.929
C05263=1147.952,127.175,-56.214,-178.916,6.760,148.928
C05264=1147.948,127.424,-56.235,-178.913,6.762,148.928
C05265=1147.942,127.673,-56.254,-178.910,6.764,148.928
C05266=1147.938,127.922,-56.273,-178.907,6.765,148.927
C05267=1147.933,128.171,-56.294,-178.905,6.767,148.927
C05268=1147.929,128.421,-56.314,-178.902,6.769,148.926
C05269=1147.923,128.669,-56.333,-178.899,6.771,148.926
C05270=1147.919,128.918,-56.353,-178.897,6.772,148.926
C05271=1147.914,129.168,-56.373,-178.894,6.774,148.925
C05272=1147.909,129.418,-56.392,-178.891,6.776,148.925
C05273=1147.904,129.666,-56.412,-178.888,6.777,148.925
C05274=1147.899,129.915,-56.432,-178.886,6.779,148.924
C05275=1147.895,130.164,-56.453,-178.883,6.781,148.924
C05276=1147.890,130.414,-56.473,-178.880,6.783,148.923
C05277=1147.885,130.663,-56.493,-178.877,6.785,148.923
C05278=1147.880,130.912,-56.512,-178.874,6.787,148.923
C05279=1147.875,131.161,-56.533,-178.871,6.788,148.922
C05280=1147.870,131.430,-56.554,-178.868,6.790,148.922
C05281=1147.865,131.699,-56.576,-178.866,6.791,148.921
C05282=1147.860,131.967,-56.597,-178.862,6.794,148.921
C05283=1147.855,132.236,-56.619,-178.860,6.796,148.920
C05284=1147.850,132.485,-56.639,-178.857,6.797,148.920
C05285=1147.845,132.734,-56.659,-178.854,6.799,148.920
C05286=1147.841,132.983,-56.679,-178.851,6.801,148.919
C05287=1147.836,133.232,-56.699,-178.849,6.803,148.919
C05288=1147.831,133.481,-56.719,-178.846,6.804,148.918
C05289=1147.826,133.730,-56.739,-178.843,6.806,148.918
C05290=1147.821,133.980,-56.760,-178.841,6.808,148.918
C05291=1147.816,134.229,-56.779,-178.837,6.810,148.917
C05292=1147.812,134.478,-56.800,-178.835,6.812,148.917
C05293=1147.807,134.726,-56.820,-178.832,6.814,148.916
C05294=1147.802,134.976,-56.839,-178.829,6.815,148.916
C05295=1147.797,135.225,-56.860,-178.826,6.817,148.916
C05296=1147.793,135.474,-56.881,-178.824,6.819,148.915
C05297=1147.788,135.724,-56.900,-178.821,6.820,148.915
C05298=1147.783,135.973,-56.921,-178.818,6.822,148.914
C05299=1147.779,136.222,-56.941,-178.816,6.824,148.914
C05300=1147.774,136.471,-56.962,-178.813,6.826,148.914
C05301=1147.769,136.721,-56.982,-178.810,6.828,148.913
C05302=1147.765,136.969,-57.002,-178.807,6.830,148.913
C05303=1147.760,137.218,-57.022,-178.804,6.832,148.913
C05304=1147.754,137.467,-57.043,-178.801,6.833,148.912
C05305=1147.750,137.717,-57.063,-178.799,6.835,148.912
C05306=1147.745,137.965,-57.083,-178.796,6.837,148.911
C05307=1147.740,138.215,-57.104,-178.793,6.838,148.911
C05308=1147.736,138.464,-57.125,-178.791,6.840,148.911
C05309=1147.731,138.713,-57.145,-178.788,6.842,148.910
C05310=1147.726,138.963,-57.165,-178.784,6.844,148.910
C05311=1147.721,139.211,-57.185,-178.782,6.846,148.909
C05312=1147.717,139.460,-57.206,-178.779,6.848,148.909
C05313=1147.712,139.710,-57.227,-178.776,6.849,148.909
C05314=1147.707,139.959,-57.247,-178.774,6.851,148.908
C05315=1147.703,140.208,-57.268,-178.771,6.853,148.908
C05316=1147.698,140.457,-57.289,-178.769,6.855,148.908
C05317=1147.693,140.706,-57.309,-178.766,6.857,148.907
C05318=1147.688,140.955,-57.329,-178.763,6.859,148.907
C05319=1147.683,141.205,-57.350,-178.760,6.861,148.907
C05320=1147.679,141.454,-57.370,-178.757,6.863,148.906
C05321=1147.674,141.703,-57.390,-178.755,6.864,148.906
C05322=1147.669,141.952,-57.411,-178.752,6.866,148.905
C05323=1147.665,142.201,-57.432,-178.749,6.868,148.905
C05324=1147.660,142.450,-57.453,-178.746,6.869,148.905
C05325=1147.655,142.699,-57.473,-178.743,6.872,148.904
C05326=1147.650,142.948,-57.494,-178.740,6.874,148.904
C05327=1147.646,143.197,-57.514,-178.738,6.875,148.903
C05328=1147.640,143.446,-57.535,-178.735,6.877,148.903
C05329=1147.636,143.695,-57.556,-178.732,6.879,148.903
C05330=1147.632,143.944,-57.576,-178.730,6.881,148.902
C05331=1147.627,144.193,-57.598,-178.726,6.883,148.902
C05332=1147.622,144.442,-57.618,-178.724,6.885,148.902
C05333=1147.617,144.691,-57.639,-178.721,6.887,148.901
C05334=1147.613,144.940,-57.659,-178.719,6.889,148.901
C05335=1147.608,145.190,-57.681,-178.716,6.890,148.901
C05336=1147.604,145.439,-57.701,-178.713,6.892,148.900
C05337=1147.598,145.688,-57.722,-178.710,6.895,148.900
C05338=1147.593,145.938,-57.743,-178.707,6.896,148.899
C05339=1147.589,146.186,-57.764,-178.704,6.898,148.899
C05340=1147.584,146.435,-57.785,-178.702,6.900,148.899
C05341=1147.579,146.684,-57.805,-178.699,6.901,148.898
C05342=1147.574,146.933,-57.826,-178.696,6.904,148.898
C05343=1147.570,147.182,-57.847,-178.693,6.906,148.898
C05344=1147.565,147.431,-57.868,-178.690,6.907,148.897
C05345=1147.560,147.681,-57.890,-178.688,6.909,148.897
C05346=1147.556,147.930,-57.910,-178.685,6.911,148.897
C05347=1147.551,148.179,-57.931,-178.683,6.913,148.896
C05348=1147.547,148.427,-57.952,-178.679,6.915,148.896
C05349=1147.542,148.677,-57.973,-178.677,6.917,148.895
C05350=1147.536,148.926,-57.994,-178.674,6.919,148.895
C05351=1147.532,149.175,-58.015,-178.671,6.921,148.895
C05352=1147.528,149.424,-58.037,-178.669,6.922,148.894
C05353=1147.522,149.673,-58.058,-178.665,6.925,148.894
C05354=1147.518,149.922,-58.078,-178.663,6.927,148.894
C05355=1147.513,150.171,-58.100,-178.660,6.929,148.893
C05356=1147.508,150.420,-58.121,-178.658,6.930,148.893
C05357=1147.504,150.669,-58.141,-178.655,6.932,148.893
C05358=1147.499,150.919,-58.163,-178.652,6.935,148.892
C05359=1147.494,151.168,-58.184,-178.649,6.936,148.892
C05360=1147.490,151.416,-58.205,-178.646,6.938,148.892
C05361=1147.485,151.665,-58.226,-178.643,6.940,148.891
C05362=1147.480,151.914,-58.248,-178.640,6.942,148.891
C05363=1147.475,152.164,-58.269,-178.638,6.944,148.891
C05364=1147.471,152.413,-58.289,-178.635,6.946,148.890
C05365=1147.466,152.662,-58.311,-178.633,6.948,148.890
C05366=1147.461,152.911,-58.332,-178.630,6.949,148.889
C05367=1147.457,153.160,-58.354,-178.627,6.952,148.889
C05368=1147.452,153.409,-58.374,-178.624,6.954,148.889
C05369=1147.447,153.658,-58.396,-178.621,6.955,148.888
C05370=1147.442,153.907,-58.417,-178.619,6.958,148.888
C05371=1147.438,154.156,-58.439,-178.616,6.960,148.888
C05372=1147.433,154.406,-58.460,-178.613,6.962,148.887
C05373=1147.429,154.654,-58.481,-178.610,6.964,148.887
C05374=1147.424,154.903,-58.503,-178.607,6.965,148.887
C05375=1147.419,155.153,-58.524,-178.604,6.968,148.886
C05376=1147.414,155.401,-58.546,-178.601,6.969,148.886
C05377=1147.409,155.651,-58.567,-178.599,6.972,148.886
C05378=1147.405,155.900,-58.589,-178.597,6.973,148.885
C05379=1147.401,156.148,-58.610,-178.593,6.976,148.885
C05380=1147.395,156.397,-58.631,-178.591,6.978,148.885
C05381=1147.391,156.646,-58.653,-178.588,6.979,148.884
C05382=1147.386,156.895,-58.675,-178.585,6.981,148.884
C05383=1147.381,157.145,-58.696,-178.582,6.984,148.884
C05384=1147.376,157.413,-58.720,-178.580,6.986,148.883
C05385=1147.371,157.682,-58.743,-178.576,6.988,148.883
C05386=1147.366,157.952,-58.766,-178.574,6.990,148.883
C05387=1147.361,158.220,-58.789,-178.570,6.992,148.882
C05388=1147.356,158.470,-58.810,-178.568,6.994,148.882
C05389=1147.351,158.718,-58.832,-178.565,6.996,148.882
C05390=1147.347,158.968,-58.854,-178.562,6.998,148.881
C05391=1147.342,159.216,-58.876,-178.559,7.000,148.881
C05392=1147.338,159.466,-58.897,-178.557,7.002,148.881
C05393=1147.333,159.715,-58.919,-178.554,7.004,148.880
C05394=1147.328,159.963,-58.940,-178.551,7.006,148.880
C05395=1147.324,160.213,-58.963,-178.548,7.008,148.880
C05396=1147.319,160.461,-58.984,-178.545,7.010,148.879
C05397=1147.314,160.711,-59.006,-178.542,7.012,148.879
C05398=1147.309,160.960,-59.027,-178.540,7.015,148.879
C05399=1147.304,161.209,-59.049,-178.537,7.016,148.878
C05400=1147.300,161.458,-59.071,-178.534,7.019,148.878
C05401=1147.295,161.707,-59.093,-178.531,7.020,148.878
C05402=1147.291,161.956,-59.115,-178.528,7.022,148.877
C05403=1147.286,162.205,-59.136,-178.526,7.024,148.877
C05404=1147.281,162.453,-59.158,-178.523,7.027,148.877
C05405=1147.277,162.703,-59.180,-178.520,7.029,148.876
C05406=1147.272,162.951,-59.202,-178.517,7.030,148.876
C05407=1147.268,163.201,-59.224,-178.515,7.033,148.876
C05408=1147.263,163.449,-59.245,-178.512,7.035,148.875
C05409=1147.259,163.699,-59.268,-178.509,7.037,148.875
C05410=1147.254,163.947,-59.289,-178.506,7.039,148.875
C05411=1147.249,164.197,-59.312,-178.503,7.041,148.874
C05412=1147.244,164.445,-59.334,-178.501,7.043,148.874
C05413=1147.240,164.695,-59.356,-178.498,7.046,148.874
C05414=1147.235,164.943,-59.377,-178.495,7.047,148.873
C05415=1147.231,165.193,-59.399,-178.492,7.049,148.873
C05416=1147.226,165.441,-59.421,-178.489,7.052,148.873
C05417=1147.221,165.690,-59.443,-178.487,7.054,148.873
C05418=1147.216,165.940,-59.465,-178.484,7.055,148.872
C05419=1147.212,166.189,-59.487,-178.481,7.058,148.872
C05420=1147.207,166.438,-59.509,-178.478,7.060,148.871
C05421=1147.202,166.687,-59.531,-178.476,7.062,148.871
C05422=1147.198,166.935,-59.554,-178.473,7.064,148.871
C05423=1147.193,167.185,-59.576,-178.470,7.066,148.871
C05424=1147.188,167.433,-59.598,-178.467,7.068,148.870
C05425=1147.184,167.683,-59.620,-178.464,7.071,148.870
C05426=1147.179,167.931,-59.642,-178.462,7.072,148.870
C05427=1147.174,168.181,-59.664,-178.459,7.074,148.869
C05428=1147.169,168.429,-59.687,-178.456,7.077,148.869
C05429=1147.165,168.678,-59.709,-178.453,7.079,148.869
C05430=1147.160,168.927,-59.730,-178.451,7.080,148.868
C05431=1147.155,169.177,-59.753,-178.447,7.083,148.868
C05432=1147.151,169.425,-59.775,-178.445,7.085,148.868
C05433=1147.146,169.674,-59.797,-178.443,7.087,148.868
C05434=1147.141,169.924,-59.820,-178.439,7.089,148.867
C05435=1147.136,170.172,-59.842,-178.437,7.091,148.867
C05436=1147.132,170.421,-59.865,-178.434,7.093,148.867
C05437=1147.127,170.670,-59.887,-178.431,7.096,148.866
C05438=1147.123,170.919,-59.909,-178.428,7.097,148.866
C05439=1147.119,171.168,-59.932,-178.425,7.100,148.866
C05440=1147.113,171.417,-59.954,-178.423,7.102,148.865
C05441=1147.109,171.666,-59.976,-178.420,7.104,148.865
C05442=1147.104,171.914,-59.998,-178.417,7.106,148.865
C05443=1147.099,172.164,-60.021,-178.415,7.108,148.865
C05444=1147.095,172.413,-60.044,-178.412,7.110,148.864
C05445=1147.090,172.661,-60.065,-178.409,7.113,148.864
C05446=1147.086,172.910,-60.089,-178.406,7.114,148.863
C05447=1147.081,173.160,-60.111,-178.403,7.117,148.863
C05448=1147.076,173.409,-60.133,-178.400,7.119,148.863
C05449=1147.072,173.657,-60.156,-178.398,7.121,148.863
C05450=1147.067,173.907,-60.179,-178.395,7.124,148.862
C05451=1147.062,174.155,-60.201,-178.392,7.125,148.862
C05452=1147.058,174.404,-60.223,-178.389,7.128,148.862
C05453=1147.053,174.653,-60.246,-178.387,7.130,148.862
C05454=1147.048,174.902,-60.268,-178.384,7.132,148.861
C05455=1147.044,175.151,-60.291,-178.381,7.134,148.861
C05456=1147.040,175.400,-60.314,-178.378,7.136,148.861
C05457=1147.034,175.649,-60.336,-178.375,7.139,148.860
C05458=1147.030,175.898,-60.359,-178.373,7.141,148.860
C05459=1147.025,176.147,-60.382,-178.370,7.142,148.860
C05460=1147.021,176.395,-60.404,-178.367,7.145,148.860
C05461=1147.016,176.645,-60.427,-178.364,7.147,148.859
C05462=1147.012,176.894,-60.450,-178.361,7.150,148.859
C05463=1147.007,177.143,-60.473,-178.359,7.152,148.859
C05464=1147.002,177.391,-60.495,-178.356,7.154,148.858
C05465=1146.997,177.640,-60.518,-178.353,7.156,148.858
C05466=1146.993,177.889,-60.541,-178.351,7.158,148.858
C05467=1146.988,178.139,-60.563,-178.347,7.161,148.858
C05468=1146.983,178.387,-60.586,-178.345,7.162,148.857
C05469=1146.979,178.636,-60.609,-178.342,7.165,148.857
C05470=1146.974,178.885,-60.633,-178.339,7.167,148.857
C05471=1146.970,179.134,-60.655,-178.336,7.170,148.857
C05472=1146.965,179.382,-60.678,-178.334,7.172,148.856
C05473=1146.960,179.631,-60.701,-178.331,7.173,148.856
C05474=1146.956,179.880,-60.724,-178.328,7.176,148.856
C05475=1146.951,180.130,-60.746,-178.325,7.178,148.855
C05476=1146.947,180.379,-60.769,-178.322,7.180,148.855
C05477=1146.942,180.627,-60.792,-178.320,7.183,148.855
C05478=1146.937,180.876,-60.815,-178.317,7.185,148.854
C05479=1146.933,181.125,-60.838,-178.314,7.187,148.854
C05480=1146.928,181.374,-60.861,-178.312,7.189,148.854
C05481=1146.924,181.623,-60.884,-178.308,7.191,148.854
C05482=1146.920,181.872,-60.907,-178.306,7.193,148.853
C05483=1146.914,182.120,-60.930,-178.303,7.196,148.853
C05484=1146.910,182.369,-60.953,-178.300,7.198,148.853
C05485=1146.905,182.618,-60.977,-178.297,7.201,148.853
C05486=1146.901,182.867,-60.999,-178.295,7.203,148.852
C05487=1146.896,183.116,-61.023,-178.291,7.205,148.852
C05488=1146.891,183.386,-61.048,-178.289,7.207,148.852
C05489=1146.886,183.655,-61.072,-178.286,7.210,148.851
C05490=1146.881,183.925,-61.097,-178.283,7.212,148.851
C05491=1146.876,184.194,-61.123,-178.279,7.215,148.851
C05492=1146.871,184.443,-61.146,-178.277,7.217,148.851
C05493=1146.867,184.692,-61.170,-178.274,7.219,148.850
C05494=1146.863,184.941,-61.193,-178.272,7.222,148.850
C05495=1146.858,185.190,-61.216,-178.268,7.224,148.850
